LIN {X 0,Y 418.5,Z 298.346,A -85,B 0,C 180,E1 -10082.888,E2 -10082.888} C_VEL
LIN {X 0,Y 418.491,Z 298.347,A -85,B 0,C 180,E1 -10086.751,E2 -10086.751} C_VEL
LIN {X 0,Y 418.4,Z 298.365,A -85,B 0,C 180,E1 -10088.695,E2 -10088.695} C_VEL
LIN {X 0,Y 418.315,Z 298.368,A -85,B 0,C 180,E1 -10091.631,E2 -10091.631} C_VEL
LIN {X 0,Y 418.303,Z 298.378,A -85,B 0,C 180,E1 -10094.597,E2 -10094.597} C_VEL
LIN {X 0,Y 418.288,Z 298.376,A -85,B 0,C 180,E1 -10097.604,E2 -10097.604} C_VEL
LIN {X 0,Y 418.25,Z 298.383,A -85,B 0,C 180,E1 -10100.663,E2 -10100.663} C_VEL
LIN {X 0,Y 418.277,Z 298.377,A -85,B 0,C 180,E1 -10103.782,E2 -10103.782} C_VEL
LIN {X 0,Y 418.311,Z 298.378,A -85,B 0,C 180,E1 -10107.071,E2 -10107.071} C_VEL
LIN {X 0,Y 418.245,Z 298.383,A -85,B 0,C 180,E1 -10110.272,E2 -10110.272} C_VEL
LIN {X 0,Y 418.249,Z 298.384,A -85,B 0,C 180,E1 -10113.677,E2 -10113.677} C_VEL
LIN {X 0,Y 418.241,Z 298.389,A -85,B 0,C 180,E1 -10117.224,E2 -10117.224} C_VEL
LIN {X 0,Y 418.247,Z 298.372,A -85,B 0,C 180,E1 -10119.683,E2 -10119.683} C_VEL
LIN {X 0,Y 418.231,Z 298.384,A -85,B 0,C 180,E1 -10122.321,E2 -10122.321} C_VEL
LIN {X 0,Y 418.237,Z 298.386,A -85,B 0,C 180,E1 -10125.109,E2 -10125.109} C_VEL
LIN {X 0,Y 418.241,Z 298.389,A -85,B 0,C 180,E1 -10127.767,E2 -10127.767} C_VEL
LIN {X 0,Y 418.247,Z 298.383,A -85,B 0,C 180,E1 -10130.621,E2 -10130.621} C_VEL
LIN {X 0,Y 418.245,Z 298.389,A -85,B 0,C 180,E1 -10133.976,E2 -10133.976} C_VEL
LIN {X 0,Y 418.26,Z 298.385,A -85,B 0,C 180,E1 -10137.156,E2 -10137.156} C_VEL
LIN {X 0,Y 418.271,Z 298.384,A -85,B 0,C 180,E1 -10140.896,E2 -10140.896} C_VEL
LIN {X 0,Y 418.35,Z 298.445,A -85,B 0,C 180,E1 -10141.77,E2 -10141.77} C_VEL
LIN {X 0,Y 421.032,Z 311.046,A -85,B 0,C 180,E1 -10144.57,E2 -10144.57} C_VEL
LIN {X 0,Y 421.704,Z 316.103,A -85,B 0,C 180,E1 -10145.639,E2 -10145.639} C_VEL
LIN {X 0,Y 420.393,Z 334.263,A -85,B 0,C 180,E1 -10149.191,E2 -10149.191} C_VEL
LIN {X 0,Y 419.959,Z 341.409,A -85,B 0,C 180,E1 -10150.575,E2 -10150.575} C_VEL
LIN {X 0,Y 424.044,Z 365.211,A -85,B 0,C 180,E1 -10151.223,E2 -10151.223} C_VEL
LIN {X 0,Y 424.504,Z 369.379,A -85,B 0,C 180,E1 -10151.321,E2 -10151.321} C_VEL
LIN {X 0,Y 423.445,Z 450.649,A -85,B 0,C 180,E1 -10152.742,E2 -10152.742} C_VEL
LIN {X 0,Y 422.844,Z 463.629,A -85,B 0,C 180,E1 -10153.152,E2 -10153.152} C_VEL
LIN {X 0,Y 422.218,Z 476.184,A -85,B 0,C 180,E1 -10153.748,E2 -10153.748} C_VEL
LIN {X 0,Y 421.378,Z 488.172,A -85,B 0,C 180,E1 -10154.522,E2 -10154.522} C_VEL
LIN {X 0,Y 420.526,Z 499.632,A -85,B 0,C 180,E1 -10155.482,E2 -10155.482} C_VEL
LIN {X 0,Y 419.746,Z 509.977,A -85,B 0,C 180,E1 -10156.566,E2 -10156.566} C_VEL
LIN {X 0,Y 419.111,Z 518.454,A -85,B 0,C 180,E1 -10157.654,E2 -10157.654} C_VEL
LIN {X 0,Y 418.291,Z 527.665,A -85,B 0,C 180,E1 -10159.104,E2 -10159.104} C_VEL
LIN {X 0,Y 417.766,Z 535.087,A -85,B 0,C 180,E1 -10160.559,E2 -10160.559} C_VEL
LIN {X 0,Y 417.368,Z 541.95,A -85,B 0,C 180,E1 -10162.258,E2 -10162.258} C_VEL
LIN {X 0,Y 417.137,Z 546.573,A -85,B 0,C 180,E1 -10163.745,E2 -10163.745} C_VEL
LIN {X 0,Y 417.107,Z 549.952,A -85,B 0,C 180,E1 -10165.167,E2 -10165.167} C_VEL
LIN {X 0,Y 417.03,Z 553.007,A -85,B 0,C 180,E1 -10167.102,E2 -10167.102} C_VEL
LIN {X 0,Y 417.07,Z 553.941,A -85,B 0,C 180,E1 -10168.068,E2 -10168.068} C_VEL
LIN {X 0,Y 417.013,Z 554.471,A -85,B 0,C 180,E1 -10169.034,E2 -10169.034} C_VEL
LIN {X 0,Y 417.027,Z 554.572,A -85,B 0,C 180,E1 -10170,E2 -10170} C_VEL
LIN {X 0,Y 417.072,Z 553.609,A -85,B 0,C 180,E1 -10171.931,E2 -10171.931} C_VEL
LIN {X 0,Y 417.061,Z 552.532,A -85,B 0,C 180,E1 -10172.897,E2 -10172.897} C_VEL
LIN {X 0,Y 417.018,Z 550.996,A -85,B 0,C 180,E1 -10173.865,E2 -10173.865} C_VEL
LIN {X 0,Y 417.119,Z 547.906,A -85,B 0,C 180,E1 -10175.317,E2 -10175.317} C_VEL
LIN {X 0,Y 417.231,Z 543.743,A -85,B 0,C 180,E1 -10176.771,E2 -10176.771} C_VEL
LIN {X 0,Y 417.481,Z 537.373,A -85,B 0,C 180,E1 -10178.47,E2 -10178.47} C_VEL
LIN {X 0,Y 417.858,Z 530.43,A -85,B 0,C 180,E1 -10179.927,E2 -10179.927} C_VEL
LIN {X 0,Y 418.281,Z 523.332,A -85,B 0,C 180,E1 -10181.141,E2 -10181.141} C_VEL
LIN {X 0,Y 418.878,Z 514.765,A -85,B 0,C 180,E1 -10182.352,E2 -10182.352} C_VEL
LIN {X 0,Y 419.513,Z 504.16,A -85,B 0,C 180,E1 -10183.564,E2 -10183.564} C_VEL
LIN {X 0,Y 420.15,Z 493.654,A -85,B 0,C 180,E1 -10184.531,E2 -10184.531} C_VEL
LIN {X 0,Y 420.876,Z 482.102,A -85,B 0,C 180,E1 -10185.372,E2 -10185.372} C_VEL
LIN {X 0,Y 421.506,Z 470.115,A -85,B 0,C 180,E1 -10186.03,E2 -10186.03} C_VEL
LIN {X 0,Y 422.019,Z 457.151,A -85,B 0,C 180,E1 -10186.538,E2 -10186.538} C_VEL
LIN {X 0,Y 422.375,Z 445.077,A -85,B 0,C 180,E1 -10186.835,E2 -10186.835} C_VEL
LIN {X 0,Y 423.05,Z 367.123,A -85,B 0,C 180,E1 -10188.161,E2 -10188.161} C_VEL
LIN {X 0,Y 419.349,Z 341.69,A -85,B 0,C 180,E1 -10188.757,E2 -10188.757} C_VEL
LIN {X 0,Y 420.441,Z 322.825,A -85,B 0,C 180,E1 -10192.351,E2 -10192.351} C_VEL
LIN {X 0,Y 420.939,Z 312.172,A -85,B 0,C 180,E1 -10194.407,E2 -10194.407} C_VEL
LIN {X 0,Y 418.487,Z 299.135,A -85,B 0,C 180,E1 -10197.117,E2 -10197.117} C_VEL
LIN {X 0,Y 418.338,Z 298.378,A -85,B 0,C 180,E1 -10197.322,E2 -10197.322} C_VEL
LIN {X 0,Y 418.239,Z 298.384,A -85,B 0,C 180,E1 -10201.019,E2 -10201.019} C_VEL
LIN {X 0,Y 418.248,Z 298.383,A -85,B 0,C 180,E1 -10203.676,E2 -10203.676} C_VEL
LIN {X 0,Y 418.238,Z 298.383,A -85,B 0,C 180,E1 -10207.223,E2 -10207.223} C_VEL
LIN {X 0,Y 418.243,Z 298.383,A -85,B 0,C 180,E1 -10209.682,E2 -10209.682} C_VEL
LIN {X 0,Y 418.228,Z 298.391,A -85,B 0,C 180,E1 -10212.32,E2 -10212.32} C_VEL
LIN {X 0,Y 418.233,Z 298.384,A -85,B 0,C 180,E1 -10215.108,E2 -10215.108} C_VEL
LIN {X 0,Y 418.238,Z 298.383,A -85,B 0,C 180,E1 -10217.766,E2 -10217.766} C_VEL
LIN {X 0,Y 418.253,Z 298.389,A -85,B 0,C 180,E1 -10220.618,E2 -10220.618} C_VEL
LIN {X 0,Y 418.24,Z 298.383,A -85,B 0,C 180,E1 -10223.975,E2 -10223.975} C_VEL
LIN {X 0,Y 418.254,Z 298.384,A -85,B 0,C 180,E1 -10227.155,E2 -10227.155} C_VEL
LIN {X 0,Y 418.265,Z 298.387,A -85,B 0,C 180,E1 -10230.895,E2 -10230.895} C_VEL
LIN {X 0,Y 418.267,Z 298.379,A -85,B 0,C 180,E1 -10234.095,E2 -10234.095} C_VEL
LIN {X 0,Y 418.234,Z 298.389,A -85,B 0,C 180,E1 -10237.263,E2 -10237.263} C_VEL
LIN {X 0,Y 418.279,Z 298.378,A -85,B 0,C 180,E1 -10240.364,E2 -10240.364} C_VEL
LIN {X 0,Y 418.313,Z 298.38,A -85,B 0,C 180,E1 -10243.404,E2 -10243.404} C_VEL
LIN {X 0,Y 418.341,Z 298.373,A -85,B 0,C 180,E1 -10246.999,E2 -10246.999} C_VEL
LIN {X 0,Y 418.336,Z 298.37,A -85,B 0,C 180,E1 -10250.328,E2 -10250.328} C_VEL
LIN {X 0,Y 418.487,Z 298.356,A -85,B 0,C 180,E1 -10253.249,E2 -10253.249} C_VEL
LIN {X 0,Y 418.333,Z 298.374,A -85,B 0,C 180,E1 -10255.181,E2 -10255.181} C_VEL
LIN {X 0,Y 418.536,Z 298.348,A -85,B 0,C 180,E1 -10258.075,E2 -10258.075} C_VEL
LIN {X 0,Y 418.665,Z 298.334,A -85,B 0,C 180,E1 -10260,E2 -10260} C_VEL
LIN {X 0,Y 418.496,Z 298.35,A -85,B 0,C 180,E1 -10262.888,E2 -10262.888} C_VEL
LIN {X 0,Y 418.452,Z 298.356,A -85,B 0,C 180,E1 -10266.52,E2 -10266.52} C_VEL
LIN {X 0,Y 418.335,Z 298.374,A -85,B 0,C 180,E1 -10269.671,E2 -10269.671} C_VEL
LIN {X 0,Y 418.341,Z 298.37,A -85,B 0,C 180,E1 -10273.001,E2 -10273.001} C_VEL
LIN {X 0,Y 418.307,Z 298.376,A -85,B 0,C 180,E1 -10276.735,E2 -10276.735} C_VEL
LIN {X 0,Y 418.265,Z 298.382,A -85,B 0,C 180,E1 -10279.79,E2 -10279.79} C_VEL
LIN {X 0,Y 418.226,Z 298.387,A -85,B 0,C 180,E1 -10282.737,E2 -10282.737} C_VEL
LIN {X 0,Y 418.256,Z 298.382,A -85,B 0,C 180,E1 -10285.905,E2 -10285.905} C_VEL
LIN {X 0,Y 418.263,Z 298.381,A -85,B 0,C 180,E1 -10289.105,E2 -10289.105} C_VEL
LIN {X 0,Y 418.252,Z 298.386,A -85,B 0,C 180,E1 -10292.844,E2 -10292.844} C_VEL
LIN {X 0,Y 418.24,Z 298.385,A -85,B 0,C 180,E1 -10296.238,E2 -10296.238} C_VEL
LIN {X 0,Y 418.24,Z 298.382,A -85,B 0,C 180,E1 -10299.683,E2 -10299.683} C_VEL
LIN {X 0,Y 418.225,Z 298.386,A -85,B 0,C 180,E1 -10302.321,E2 -10302.321} C_VEL
LIN {X 0,Y 418.231,Z 298.389,A -85,B 0,C 180,E1 -10305.109,E2 -10305.109} C_VEL
LIN {X 0,Y 418.219,Z 298.386,A -85,B 0,C 180,E1 -10307.765,E2 -10307.765} C_VEL
LIN {X 0,Y 418.236,Z 298.386,A -85,B 0,C 180,E1 -10311.557,E2 -10311.557} C_VEL
LIN {X 0,Y 418.254,Z 298.388,A -85,B 0,C 180,E1 -10315.159,E2 -10315.159} C_VEL
LIN {X 0,Y 418.242,Z 298.388,A -85,B 0,C 180,E1 -10317.472,E2 -10317.472} C_VEL
LIN {X 0,Y 418.258,Z 298.382,A -85,B 0,C 180,E1 -10320.898,E2 -10320.898} C_VEL
LIN {X 0,Y 418.221,Z 298.386,A -85,B 0,C 180,E1 -10324.093,E2 -10324.093} C_VEL
LIN {X 0,Y 418.225,Z 298.388,A -85,B 0,C 180,E1 -10327.264,E2 -10327.264} C_VEL
LIN {X 0,Y 418.281,Z 298.378,A -85,B 0,C 180,E1 -10330.365,E2 -10330.365} C_VEL
LIN {X 0,Y 418.314,Z 298.377,A -85,B 0,C 180,E1 -10333.405,E2 -10333.405} C_VEL
LIN {X 0,Y 418.344,Z 298.373,A -85,B 0,C 180,E1 -10337,E2 -10337} C_VEL
LIN {X 0,Y 418.402,Z 298.509,A -85,B 0,C 180,E1 -10338.218,E2 -10338.218} C_VEL
LIN {X 0,Y 419.848,Z 307.982,A -85,B 0,C 180,E1 -10340.364,E2 -10340.364} C_VEL
LIN {X 0,Y 419.769,Z 312.482,A -85,B 0,C 180,E1 -10341.334,E2 -10341.334} C_VEL
LIN {X 0,Y 423.405,Z 332.436,A -85,B 0,C 180,E1 -10341.834,E2 -10341.834} C_VEL
LIN {X 0,Y 422.377,Z 420.161,A -85,B 0,C 180,E1 -10343.342,E2 -10343.342} C_VEL
LIN {X 0,Y 422.005,Z 433.941,A -85,B 0,C 180,E1 -10343.786,E2 -10343.786} C_VEL
LIN {X 0,Y 421.617,Z 446.275,A -85,B 0,C 180,E1 -10344.38,E2 -10344.38} C_VEL
LIN {X 0,Y 421.232,Z 455.15,A -85,B 0,C 180,E1 -10344.942,E2 -10344.942} C_VEL
LIN {X 0,Y 420.359,Z 458.68,A -85,B 0,C 180,E1 -10345.169,E2 -10345.169} C_VEL
LIN {X 0,Y 417.152,Z 464.137,A -85,B 0,C 180,E1 -10345.503,E2 -10345.503} C_VEL
LIN {X 0,Y 413.955,Z 469.396,A -85,B 0,C 180,E1 -10345.888,E2 -10345.888} C_VEL
LIN {X 0,Y 413.101,Z 472.61,A -85,B 0,C 180,E1 -10346.19,E2 -10346.19} C_VEL
LIN {X 0,Y 412.334,Z 482.525,A -85,B 0,C 180,E1 -10347.314,E2 -10347.314} C_VEL
LIN {X 0,Y 411.859,Z 491.264,A -85,B 0,C 180,E1 -10348.534,E2 -10348.534} C_VEL
LIN {X 0,Y 411.253,Z 499.825,A -85,B 0,C 180,E1 -10350,E2 -10350} C_VEL
LIN {X 0,Y 410.769,Z 506.671,A -85,B 0,C 180,E1 -10351.471,E2 -10351.471} C_VEL
LIN {X 0,Y 410.451,Z 512.158,A -85,B 0,C 180,E1 -10352.945,E2 -10352.945} C_VEL
LIN {X 0,Y 410.172,Z 516.476,A -85,B 0,C 180,E1 -10354.422,E2 -10354.422} C_VEL
LIN {X 0,Y 410.15,Z 519.723,A -85,B 0,C 180,E1 -10355.901,E2 -10355.901} C_VEL
LIN {X 0,Y 410.05,Z 521.347,A -85,B 0,C 180,E1 -10356.891,E2 -10356.891} C_VEL
LIN {X 0,Y 409.941,Z 522.573,A -85,B 0,C 180,E1 -10357.883,E2 -10357.883} C_VEL
LIN {X 0,Y 409.863,Z 523.362,A -85,B 0,C 180,E1 -10358.878,E2 -10358.878} C_VEL
LIN {X 0,Y 409.93,Z 523.73,A -85,B 0,C 180,E1 -10360.871,E2 -10360.871} C_VEL
LIN {X 0,Y 409.993,Z 523.009,A -85,B 0,C 180,E1 -10362.291,E2 -10362.291} C_VEL
LIN {X 0,Y 410.048,Z 521.225,A -85,B 0,C 180,E1 -10363.884,E2 -10363.884} C_VEL
LIN {X 0,Y 410.293,Z 518.521,A -85,B 0,C 180,E1 -10365.397,E2 -10365.397} C_VEL
LIN {X 0,Y 410.547,Z 514.751,A -85,B 0,C 180,E1 -10366.919,E2 -10366.919} C_VEL
LIN {X 0,Y 410.942,Z 509.796,A -85,B 0,C 180,E1 -10368.445,E2 -10368.445} C_VEL
LIN {X 0,Y 411.611,Z 502.906,A -85,B 0,C 180,E1 -10370.101,E2 -10370.101} C_VEL
LIN {X 0,Y 412.178,Z 495.548,A -85,B 0,C 180,E1 -10371.506,E2 -10371.506} C_VEL
LIN {X 0,Y 412.961,Z 487.353,A -85,B 0,C 180,E1 -10372.779,E2 -10372.779} C_VEL
LIN {X 0,Y 413.852,Z 477.278,A -85,B 0,C 180,E1 -10374.052,E2 -10374.052} C_VEL
LIN {X 0,Y 414.666,Z 467.31,A -85,B 0,C 180,E1 -10375.069,E2 -10375.069} C_VEL
LIN {X 0,Y 415.429,Z 456.392,A -85,B 0,C 180,E1 -10375.96,E2 -10375.96} C_VEL
LIN {X 0,Y 416.125,Z 444.455,A -85,B 0,C 180,E1 -10376.713,E2 -10376.713} C_VEL
LIN {X 0,Y 416.599,Z 431.865,A -85,B 0,C 180,E1 -10377.3,E2 -10377.3} C_VEL
LIN {X 0,Y 416.859,Z 420.649,A -85,B 0,C 180,E1 -10377.656,E2 -10377.656} C_VEL
LIN {X 0,Y 418.259,Z 333.539,A -85,B 0,C 180,E1 -10379.19,E2 -10379.19} C_VEL
LIN {X 0,Y 413.571,Z 313.012,A -85,B 0,C 180,E1 -10379.833,E2 -10379.833} C_VEL
LIN {X 0,Y 413.27,Z 309.221,A -85,B 0,C 180,E1 -10380.676,E2 -10380.676} C_VEL
LIN {X 0,Y 411.221,Z 299.263,A -85,B 0,C 180,E1 -10383.068,E2 -10383.068} C_VEL
LIN {X 0,Y 411.192,Z 299.263,A -85,B 0,C 180,E1 -10386.553,E2 -10386.553} C_VEL
LIN {X 0,Y 411.21,Z 299.263,A -85,B 0,C 180,E1 -10389.728,E2 -10389.728} C_VEL
LIN {X 0,Y 411.172,Z 299.267,A -85,B 0,C 180,E1 -10393.134,E2 -10393.134} C_VEL
LIN {X 0,Y 411.167,Z 299.266,A -85,B 0,C 180,E1 -10395.881,E2 -10395.881} C_VEL
LIN {X 0,Y 411.163,Z 299.27,A -85,B 0,C 180,E1 -10398.772,E2 -10398.772} C_VEL
LIN {X 0,Y 411.205,Z 299.257,A -85,B 0,C 180,E1 -10401.831,E2 -10401.831} C_VEL
LIN {X 0,Y 411.21,Z 299.261,A -85,B 0,C 180,E1 -10405.122,E2 -10405.122} C_VEL
LIN {X 0,Y 411.165,Z 299.26,A -85,B 0,C 180,E1 -10408.003,E2 -10408.003} C_VEL
LIN {X 0,Y 411.217,Z 299.256,A -85,B 0,C 180,E1 -10411.41,E2 -10411.41} C_VEL
LIN {X 0,Y 411.236,Z 299.255,A -85,B 0,C 180,E1 -10413.619,E2 -10413.619} C_VEL
LIN {X 0,Y 411.196,Z 299.256,A -85,B 0,C 180,E1 -10416.852,E2 -10416.852} C_VEL
LIN {X 0,Y 411.214,Z 299.253,A -85,B 0,C 180,E1 -10420.051,E2 -10420.051} C_VEL
LIN {X 0,Y 411.262,Z 299.256,A -85,B 0,C 180,E1 -10423.131,E2 -10423.131} C_VEL
LIN {X 0,Y 411.305,Z 299.248,A -85,B 0,C 180,E1 -10426.896,E2 -10426.896} C_VEL
LIN {X 0,Y 411.292,Z 299.251,A -85,B 0,C 180,E1 -10430.161,E2 -10430.161} C_VEL
LIN {X 0,Y 411.482,Z 299.226,A -85,B 0,C 180,E1 -10432.147,E2 -10432.147} C_VEL
LIN {X 0,Y 411.471,Z 299.229,A -85,B 0,C 180,E1 -10434.118,E2 -10434.118} C_VEL
LIN {X 0,Y 411.511,Z 299.221,A -85,B 0,C 180,E1 -10438.043,E2 -10438.043} C_VEL
LIN {X 0,Y 411.64,Z 299.21,A -85,B 0,C 180,E1 -10440,E2 -10440} C_VEL
LIN {X 0,Y 411.457,Z 299.223,A -85,B 0,C 180,E1 -10442.937,E2 -10442.937} C_VEL
LIN {X 0,Y 411.458,Z 299.222,A -85,B 0,C 180,E1 -10446.867,E2 -10446.867} C_VEL
LIN {X 0,Y 411.354,Z 299.241,A -85,B 0,C 180,E1 -10448.845,E2 -10448.845} C_VEL
LIN {X 0,Y 411.283,Z 299.245,A -85,B 0,C 180,E1 -10451.833,E2 -10451.833} C_VEL
LIN {X 0,Y 411.26,Z 299.252,A -85,B 0,C 180,E1 -10454.853,E2 -10454.853} C_VEL
LIN {X 0,Y 411.253,Z 299.253,A -85,B 0,C 180,E1 -10457.915,E2 -10457.915} C_VEL
LIN {X 0,Y 411.197,Z 299.263,A -85,B 0,C 180,E1 -10461.034,E2 -10461.034} C_VEL
LIN {X 0,Y 411.221,Z 299.257,A -85,B 0,C 180,E1 -10464.216,E2 -10464.216} C_VEL
LIN {X 0,Y 411.26,Z 299.253,A -85,B 0,C 180,E1 -10467.478,E2 -10467.478} C_VEL
LIN {X 0,Y 411.19,Z 299.268,A -85,B 0,C 180,E1 -10470.848,E2 -10470.848} C_VEL
LIN {X 0,Y 411.206,Z 299.26,A -85,B 0,C 180,E1 -10474.334,E2 -10474.334} C_VEL
LIN {X 0,Y 411.194,Z 299.261,A -85,B 0,C 180,E1 -10477.974,E2 -10477.974} C_VEL
LIN {X 0,Y 411.165,Z 299.255,A -85,B 0,C 180,E1 -10481.229,E2 -10481.229} C_VEL
LIN {X 0,Y 411.177,Z 299.262,A -85,B 0,C 180,E1 -10484.491,E2 -10484.491} C_VEL
LIN {X 0,Y 411.178,Z 299.265,A -85,B 0,C 180,E1 -10488.195,E2 -10488.195} C_VEL
LIN {X 0,Y 411.212,Z 299.259,A -85,B 0,C 180,E1 -10490.775,E2 -10490.775} C_VEL
LIN {X 0,Y 411.2,Z 299.263,A -85,B 0,C 180,E1 -10494.471,E2 -10494.471} C_VEL
LIN {X 0,Y 411.21,Z 299.263,A -85,B 0,C 180,E1 -10496.873,E2 -10496.873} C_VEL
LIN {X 0,Y 411.235,Z 299.26,A -85,B 0,C 180,E1 -10500.644,E2 -10500.644} C_VEL
LIN {X 0,Y 411.293,Z 299.263,A -85,B 0,C 180,E1 -10501.416,E2 -10501.416} C_VEL
LIN {X 0,Y 413.882,Z 311.315,A -85,B 0,C 180,E1 -10504.156,E2 -10504.156} C_VEL
LIN {X 0,Y 414.812,Z 317.388,A -85,B 0,C 180,E1 -10505.475,E2 -10505.475} C_VEL
LIN {X 0,Y 413.452,Z 335.534,A -85,B 0,C 180,E1 -10509.086,E2 -10509.086} C_VEL
LIN {X 0,Y 413.097,Z 341.103,A -85,B 0,C 180,E1 -10510.184,E2 -10510.184} C_VEL
LIN {X 0,Y 417.21,Z 364.546,A -85,B 0,C 180,E1 -10510.848,E2 -10510.848} C_VEL
LIN {X 0,Y 417.876,Z 371.311,A -85,B 0,C 180,E1 -10511.007,E2 -10511.007} C_VEL
LIN {X 0,Y 416.813,Z 449.726,A -85,B 0,C 180,E1 -10512.395,E2 -10512.395} C_VEL
LIN {X 0,Y 416.15,Z 462.924,A -85,B 0,C 180,E1 -10512.81,E2 -10512.81} C_VEL
LIN {X 0,Y 415.502,Z 475.585,A -85,B 0,C 180,E1 -10513.415,E2 -10513.415} C_VEL
LIN {X 0,Y 414.683,Z 486.873,A -85,B 0,C 180,E1 -10514.14,E2 -10514.14} C_VEL
LIN {X 0,Y 413.765,Z 498.523,A -85,B 0,C 180,E1 -10515.113,E2 -10515.113} C_VEL
LIN {X 0,Y 412.88,Z 509.01,A -85,B 0,C 180,E1 -10516.213,E2 -10516.213} C_VEL
LIN {X 0,Y 412.154,Z 518.486,A -85,B 0,C 180,E1 -10517.443,E2 -10517.443} C_VEL
LIN {X 0,Y 411.307,Z 527.627,A -85,B 0,C 180,E1 -10518.917,E2 -10518.917} C_VEL
LIN {X 0,Y 410.741,Z 535.006,A -85,B 0,C 180,E1 -10520.396,E2 -10520.396} C_VEL
LIN {X 0,Y 410.322,Z 541.816,A -85,B 0,C 180,E1 -10522.124,E2 -10522.124} C_VEL
LIN {X 0,Y 410.043,Z 546.76,A -85,B 0,C 180,E1 -10523.776,E2 -10523.776} C_VEL
LIN {X 0,Y 410.019,Z 549.761,A -85,B 0,C 180,E1 -10525.083,E2 -10525.083} C_VEL
LIN {X 0,Y 409.928,Z 552.786,A -85,B 0,C 180,E1 -10527.051,E2 -10527.051} C_VEL
LIN {X 0,Y 409.997,Z 553.709,A -85,B 0,C 180,E1 -10528.035,E2 -10528.035} C_VEL
LIN {X 0,Y 409.938,Z 554.216,A -85,B 0,C 180,E1 -10529.017,E2 -10529.017} C_VEL
LIN {X 0,Y 409.948,Z 554.301,A -85,B 0,C 180,E1 -10530,E2 -10530} C_VEL
LIN {X 0,Y 410.001,Z 553.314,A -85,B 0,C 180,E1 -10531.964,E2 -10531.964} C_VEL
LIN {X 0,Y 409.959,Z 552.213,A -85,B 0,C 180,E1 -10532.948,E2 -10532.948} C_VEL
LIN {X 0,Y 409.937,Z 550.661,A -85,B 0,C 180,E1 -10533.932,E2 -10533.932} C_VEL
LIN {X 0,Y 410.014,Z 547.54,A -85,B 0,C 180,E1 -10535.409,E2 -10535.409} C_VEL
LIN {X 0,Y 410.163,Z 543.347,A -85,B 0,C 180,E1 -10536.888,E2 -10536.888} C_VEL
LIN {X 0,Y 410.413,Z 536.942,A -85,B 0,C 180,E1 -10538.617,E2 -10538.617} C_VEL
LIN {X 0,Y 410.8,Z 529.958,A -85,B 0,C 180,E1 -10540.099,E2 -10540.099} C_VEL
LIN {X 0,Y 411.381,Z 521.191,A -85,B 0,C 180,E1 -10541.58,E2 -10541.58} C_VEL
LIN {X 0,Y 411.996,Z 512.2,A -85,B 0,C 180,E1 -10542.812,E2 -10542.812} C_VEL
LIN {X 0,Y 412.588,Z 503.016,A -85,B 0,C 180,E1 -10543.847,E2 -10543.847} C_VEL
LIN {X 0,Y 413.22,Z 492.899,A -85,B 0,C 180,E1 -10544.78,E2 -10544.78} C_VEL
LIN {X 0,Y 414,Z 481.167,A -85,B 0,C 180,E1 -10545.634,E2 -10545.634} C_VEL
LIN {X 0,Y 414.609,Z 468.943,A -85,B 0,C 180,E1 -10546.304,E2 -10546.304} C_VEL
LIN {X 0,Y 415.215,Z 455.622,A -85,B 0,C 180,E1 -10546.817,E2 -10546.817} C_VEL
LIN {X 0,Y 415.558,Z 442.471,A -85,B 0,C 180,E1 -10547.12,E2 -10547.12} C_VEL
LIN {X 0,Y 416.225,Z 367.94,A -85,B 0,C 180,E1 -10548.406,E2 -10548.406} C_VEL
LIN {X 0,Y 412.405,Z 341.35,A -85,B 0,C 180,E1 -10549.053,E2 -10549.053} C_VEL
LIN {X 0,Y 413.456,Z 323.637,A -85,B 0,C 180,E1 -10552.485,E2 -10552.485} C_VEL
LIN {X 0,Y 414.045,Z 314.324,A -85,B 0,C 180,E1 -10554.306,E2 -10554.306} C_VEL
LIN {X 0,Y 412.136,Z 303.43,A -85,B 0,C 180,E1 -10556.591,E2 -10556.591} C_VEL
LIN {X 0,Y 411.314,Z 299.253,A -85,B 0,C 180,E1 -10557.507,E2 -10557.507} C_VEL
LIN {X 0,Y 411.189,Z 299.264,A -85,B 0,C 180,E1 -10560.847,E2 -10560.847} C_VEL
LIN {X 0,Y 411.206,Z 299.265,A -85,B 0,C 180,E1 -10564.333,E2 -10564.333} C_VEL
LIN {X 0,Y 411.19,Z 299.264,A -85,B 0,C 180,E1 -10567.973,E2 -10567.973} C_VEL
LIN {X 0,Y 411.162,Z 299.264,A -85,B 0,C 180,E1 -10571.228,E2 -10571.228} C_VEL
LIN {X 0,Y 411.174,Z 299.271,A -85,B 0,C 180,E1 -10574.49,E2 -10574.49} C_VEL
LIN {X 0,Y 411.175,Z 299.266,A -85,B 0,C 180,E1 -10578.194,E2 -10578.194} C_VEL
LIN {X 0,Y 411.217,Z 299.264,A -85,B 0,C 180,E1 -10580.775,E2 -10580.775} C_VEL
LIN {X 0,Y 411.195,Z 299.264,A -85,B 0,C 180,E1 -10584.471,E2 -10584.471} C_VEL
LIN {X 0,Y 411.204,Z 299.266,A -85,B 0,C 180,E1 -10586.873,E2 -10586.873} C_VEL
LIN {X 0,Y 411.229,Z 299.26,A -85,B 0,C 180,E1 -10590.644,E2 -10590.644} C_VEL
LIN {X 0,Y 411.234,Z 299.256,A -85,B 0,C 180,E1 -10593.619,E2 -10593.619} C_VEL
LIN {X 0,Y 411.199,Z 299.264,A -85,B 0,C 180,E1 -10596.852,E2 -10596.852} C_VEL
LIN {X 0,Y 411.21,Z 299.258,A -85,B 0,C 180,E1 -10600.05,E2 -10600.05} C_VEL
LIN {X 0,Y 411.259,Z 299.258,A -85,B 0,C 180,E1 -10603.131,E2 -10603.131} C_VEL
LIN {X 0,Y 411.301,Z 299.249,A -85,B 0,C 180,E1 -10606.895,E2 -10606.895} C_VEL
LIN {X 0,Y 411.288,Z 299.249,A -85,B 0,C 180,E1 -10610.161,E2 -10610.161} C_VEL
LIN {X 0,Y 411.45,Z 299.231,A -85,B 0,C 180,E1 -10613.133,E2 -10613.133} C_VEL
LIN {X 0,Y 411.304,Z 299.249,A -85,B 0,C 180,E1 -10615.099,E2 -10615.099} C_VEL
LIN {X 0,Y 411.505,Z 299.225,A -85,B 0,C 180,E1 -10618.042,E2 -10618.042} C_VEL
LIN {X 0,Y 411.634,Z 299.21,A -85,B 0,C 180,E1 -10620,E2 -10620} C_VEL
LIN {X 0,Y 411.453,Z 299.228,A -85,B 0,C 180,E1 -10622.937,E2 -10622.937} C_VEL
LIN {X 0,Y 411.417,Z 299.234,A -85,B 0,C 180,E1 -10626.517,E2 -10626.517} C_VEL
LIN {X 0,Y 411.287,Z 299.254,A -85,B 0,C 180,E1 -10629.839,E2 -10629.839} C_VEL
LIN {X 0,Y 411.3,Z 299.247,A -85,B 0,C 180,E1 -10633.104,E2 -10633.104} C_VEL
LIN {X 0,Y 411.252,Z 299.254,A -85,B 0,C 180,E1 -10636.889,E2 -10636.889} C_VEL
LIN {X 0,Y 411.225,Z 299.26,A -85,B 0,C 180,E1 -10639.987,E2 -10639.987} C_VEL
LIN {X 0,Y 411.19,Z 299.261,A -85,B 0,C 180,E1 -10643.148,E2 -10643.148} C_VEL
LIN {X 0,Y 411.228,Z 299.263,A -85,B 0,C 180,E1 -10646.381,E2 -10646.381} C_VEL
LIN {X 0,Y 411.195,Z 299.26,A -85,B 0,C 180,E1 -10649.713,E2 -10649.713} C_VEL
LIN {X 0,Y 411.201,Z 299.261,A -85,B 0,C 180,E1 -10653.156,E2 -10653.156} C_VEL
LIN {X 0,Y 411.187,Z 299.267,A -85,B 0,C 180,E1 -10656.553,E2 -10656.553} C_VEL
LIN {X 0,Y 411.204,Z 299.259,A -85,B 0,C 180,E1 -10659.727,E2 -10659.727} C_VEL
LIN {X 0,Y 411.168,Z 299.268,A -85,B 0,C 180,E1 -10663.134,E2 -10663.134} C_VEL
LIN {X 0,Y 411.16,Z 299.264,A -85,B 0,C 180,E1 -10665.882,E2 -10665.882} C_VEL
LIN {X 0,Y 411.146,Z 299.27,A -85,B 0,C 180,E1 -10668.774,E2 -10668.774} C_VEL
LIN {X 0,Y 411.184,Z 299.262,A -85,B 0,C 180,E1 -10672.026,E2 -10672.026} C_VEL
LIN {X 0,Y 411.201,Z 299.262,A -85,B 0,C 180,E1 -10675.667,E2 -10675.667} C_VEL
LIN {X 0,Y 411.186,Z 299.267,A -85,B 0,C 180,E1 -10679.153,E2 -10679.153} C_VEL
LIN {X 0,Y 411.174,Z 299.271,A -85,B 0,C 180,E1 -10681.407,E2 -10681.407} C_VEL
LIN {X 0,Y 411.185,Z 299.263,A -85,B 0,C 180,E1 -10684.942,E2 -10684.942} C_VEL
LIN {X 0,Y 411.201,Z 299.263,A -85,B 0,C 180,E1 -10687.914,E2 -10687.914} C_VEL
LIN {X 0,Y 411.216,Z 299.259,A -85,B 0,C 180,E1 -10691.052,E2 -10691.052} C_VEL
LIN {X 0,Y 411.252,Z 299.258,A -85,B 0,C 180,E1 -10694.132,E2 -10694.132} C_VEL
LIN {X 0,Y 411.349,Z 299.328,A -85,B 0,C 180,E1 -10698.013,E2 -10698.013} C_VEL
LIN {X 0,Y 412.876,Z 308.819,A -85,B 0,C 180,E1 -10700.2,E2 -10700.2} C_VEL
LIN {X 0,Y 412.847,Z 313.009,A -85,B 0,C 180,E1 -10701.069,E2 -10701.069} C_VEL
LIN {X 0,Y 416.598,Z 333.572,A -85,B 0,C 180,E1 -10701.586,E2 -10701.586} C_VEL
LIN {X 0,Y 415.512,Z 420.703,A -85,B 0,C 180,E1 -10703.109,E2 -10703.109} C_VEL
LIN {X 0,Y 415.124,Z 434.395,A -85,B 0,C 180,E1 -10703.561,E2 -10703.561} C_VEL
LIN {X 0,Y 414.715,Z 446.675,A -85,B 0,C 180,E1 -10704.165,E2 -10704.165} C_VEL
LIN {X 0,Y 414.16,Z 457.694,A -85,B 0,C 180,E1 -10704.889,E2 -10704.889} C_VEL
LIN {X 0,Y 413.359,Z 467.932,A -85,B 0,C 180,E1 -10705.735,E2 -10705.735} C_VEL
LIN {X 0,Y 413.101,Z 472.61,A -85,B 0,C 180,E1 -10706.19,E2 -10706.19} C_VEL
LIN {X 0,Y 412.195,Z 477.351,A -85,B 0,C 180,E1 -10706.68,E2 -10706.68} C_VEL
LIN {X 0,Y 408.853,Z 484.704,A -85,B 0,C 180,E1 -10707.491,E2 -10707.491} C_VEL
LIN {X 0,Y 405.502,Z 491.482,A -85,B 0,C 180,E1 -10708.387,E2 -10708.387} C_VEL
LIN {X 0,Y 404.583,Z 495.318,A -85,B 0,C 180,E1 -10708.998,E2 -10708.998} C_VEL
LIN {X 0,Y 403.946,Z 503.177,A -85,B 0,C 180,E1 -10710.499,E2 -10710.499} C_VEL
LIN {X 0,Y 403.538,Z 509.415,A -85,B 0,C 180,E1 -10711.996,E2 -10711.996} C_VEL
LIN {X 0,Y 403.28,Z 514.384,A -85,B 0,C 180,E1 -10713.497,E2 -10713.497} C_VEL
LIN {X 0,Y 403.106,Z 518.239,A -85,B 0,C 180,E1 -10715.001,E2 -10715.001} C_VEL
LIN {X 0,Y 403.074,Z 520.846,A -85,B 0,C 180,E1 -10716.358,E2 -10716.358} C_VEL
LIN {X 0,Y 402.836,Z 522.968,A -85,B 0,C 180,E1 -10718.023,E2 -10718.023} C_VEL
LIN {X 0,Y 402.753,Z 524.028,A -85,B 0,C 180,E1 -10720.05,E2 -10720.05} C_VEL
LIN {X 0,Y 402.837,Z 523.975,A -85,B 0,C 180,E1 -10721.064,E2 -10721.064} C_VEL
LIN {X 0,Y 402.925,Z 523.275,A -85,B 0,C 180,E1 -10722.373,E2 -10722.373} C_VEL
LIN {X 0,Y 402.986,Z 521.296,A -85,B 0,C 180,E1 -10724.132,E2 -10724.132} C_VEL
LIN {X 0,Y 403.263,Z 518.501,A -85,B 0,C 180,E1 -10725.672,E2 -10725.672} C_VEL
LIN {X 0,Y 403.559,Z 514.633,A -85,B 0,C 180,E1 -10727.221,E2 -10727.221} C_VEL
LIN {X 0,Y 404.018,Z 509.574,A -85,B 0,C 180,E1 -10728.773,E2 -10728.773} C_VEL
LIN {X 0,Y 404.659,Z 503.152,A -85,B 0,C 180,E1 -10730.326,E2 -10730.326} C_VEL
LIN {X 0,Y 405.352,Z 495.012,A -85,B 0,C 180,E1 -10731.887,E2 -10731.887} C_VEL
LIN {X 0,Y 406.195,Z 486.657,A -85,B 0,C 180,E1 -10733.18,E2 -10733.18} C_VEL
LIN {X 0,Y 407.152,Z 476.377,A -85,B 0,C 180,E1 -10734.474,E2 -10734.474} C_VEL
LIN {X 0,Y 407.997,Z 466.069,A -85,B 0,C 180,E1 -10735.508,E2 -10735.508} C_VEL
LIN {X 0,Y 408.836,Z 454.76,A -85,B 0,C 180,E1 -10736.411,E2 -10736.411} C_VEL
LIN {X 0,Y 409.549,Z 442.103,A -85,B 0,C 180,E1 -10737.187,E2 -10737.187} C_VEL
LIN {X 0,Y 410.004,Z 429.317,A -85,B 0,C 180,E1 -10737.742,E2 -10737.742} C_VEL
LIN {X 0,Y 410.324,Z 419.457,A -85,B 0,C 180,E1 -10738.031,E2 -10738.031} C_VEL
LIN {X 0,Y 411.721,Z 334.697,A -85,B 0,C 180,E1 -10739.538,E2 -10739.538} C_VEL
LIN {X 0,Y 407.005,Z 314.386,A -85,B 0,C 180,E1 -10740.197,E2 -10740.197} C_VEL
LIN {X 0,Y 406.707,Z 313.102,A -85,B 0,C 180,E1 -10740.254,E2 -10740.254} C_VEL
LIN {X 0,Y 405.303,Z 305.327,A -85,B 0,C 180,E1 -10742.124,E2 -10742.124} C_VEL
LIN {X 0,Y 404.168,Z 300.142,A -85,B 0,C 180,E1 -10743.419,E2 -10743.419} C_VEL
LIN {X 0,Y 404.141,Z 300.146,A -85,B 0,C 180,E1 -10746.246,E2 -10746.246} C_VEL
LIN {X 0,Y 404.152,Z 300.145,A -85,B 0,C 180,E1 -10748.757,E2 -10748.757} C_VEL
LIN {X 0,Y 404.122,Z 300.144,A -85,B 0,C 180,E1 -10751.6,E2 -10751.6} C_VEL
LIN {X 0,Y 404.144,Z 300.142,A -85,B 0,C 180,E1 -10754.522,E2 -10754.522} C_VEL
LIN {X 0,Y 404.136,Z 300.142,A -85,B 0,C 180,E1 -10757.296,E2 -10757.296} C_VEL
LIN {X 0,Y 404.168,Z 300.136,A -85,B 0,C 180,E1 -10759.955,E2 -10759.955} C_VEL
LIN {X 0,Y 404.136,Z 300.142,A -85,B 0,C 180,E1 -10763.125,E2 -10763.125} C_VEL
LIN {X 0,Y 404.144,Z 300.136,A -85,B 0,C 180,E1 -10766.188,E2 -10766.188} C_VEL
LIN {X 0,Y 404.145,Z 300.135,A -85,B 0,C 180,E1 -10769.715,E2 -10769.715} C_VEL
LIN {X 0,Y 404.194,Z 300.13,A -85,B 0,C 180,E1 -10773.123,E2 -10773.123} C_VEL
LIN {X 0,Y 404.173,Z 300.135,A -85,B 0,C 180,E1 -10775.334,E2 -10775.334} C_VEL
LIN {X 0,Y 404.137,Z 300.139,A -85,B 0,C 180,E1 -10778.581,E2 -10778.581} C_VEL
LIN {X 0,Y 404.209,Z 300.135,A -85,B 0,C 180,E1 -10781.762,E2 -10781.762} C_VEL
LIN {X 0,Y 404.205,Z 300.128,A -85,B 0,C 180,E1 -10784.882,E2 -10784.882} C_VEL
LIN {X 0,Y 404.255,Z 300.126,A -85,B 0,C 180,E1 -10787.959,E2 -10787.959} C_VEL
LIN {X 0,Y 404.433,Z 300.104,A -85,B 0,C 180,E1 -10792.1,E2 -10792.1} C_VEL
LIN {X 0,Y 404.42,Z 300.106,A -85,B 0,C 180,E1 -10794.015,E2 -10794.015} C_VEL
LIN {X 0,Y 404.48,Z 300.096,A -85,B 0,C 180,E1 -10798.009,E2 -10798.009} C_VEL
LIN {X 0,Y 404.609,Z 300.086,A -85,B 0,C 180,E1 -10800,E2 -10800} C_VEL
LIN {X 0,Y 404.415,Z 300.1,A -85,B 0,C 180,E1 -10802.989,E2 -10802.989} C_VEL
LIN {X 0,Y 404.41,Z 300.099,A -85,B 0,C 180,E1 -10806.988,E2 -10806.988} C_VEL
LIN {X 0,Y 404.258,Z 300.127,A -85,B 0,C 180,E1 -10810.012,E2 -10810.012} C_VEL
LIN {X 0,Y 404.267,Z 300.123,A -85,B 0,C 180,E1 -10813.212,E2 -10813.212} C_VEL
LIN {X 0,Y 404.216,Z 300.131,A -85,B 0,C 180,E1 -10817.007,E2 -10817.007} C_VEL
LIN {X 0,Y 404.164,Z 300.136,A -85,B 0,C 180,E1 -10820.352,E2 -10820.352} C_VEL
LIN {X 0,Y 404.164,Z 300.135,A -85,B 0,C 180,E1 -10823.575,E2 -10823.575} C_VEL
LIN {X 0,Y 404.184,Z 300.134,A -85,B 0,C 180,E1 -10825.767,E2 -10825.767} C_VEL
LIN {X 0,Y 404.196,Z 300.131,A -85,B 0,C 180,E1 -10828,E2 -10828} C_VEL
LIN {X 0,Y 404.14,Z 300.139,A -85,B 0,C 180,E1 -10831.558,E2 -10831.558} C_VEL
LIN {X 0,Y 404.185,Z 300.138,A -85,B 0,C 180,E1 -10835.016,E2 -10835.016} C_VEL
LIN {X 0,Y 404.153,Z 300.14,A -85,B 0,C 180,E1 -10838.757,E2 -10838.757} C_VEL
LIN {X 0,Y 404.124,Z 300.137,A -85,B 0,C 180,E1 -10841.6,E2 -10841.6} C_VEL
LIN {X 0,Y 404.147,Z 300.138,A -85,B 0,C 180,E1 -10844.522,E2 -10844.522} C_VEL
LIN {X 0,Y 404.138,Z 300.144,A -85,B 0,C 180,E1 -10847.296,E2 -10847.296} C_VEL
LIN {X 0,Y 404.171,Z 300.139,A -85,B 0,C 180,E1 -10849.956,E2 -10849.956} C_VEL
LIN {X 0,Y 404.138,Z 300.138,A -85,B 0,C 180,E1 -10853.125,E2 -10853.125} C_VEL
LIN {X 0,Y 404.147,Z 300.145,A -85,B 0,C 180,E1 -10856.188,E2 -10856.188} C_VEL
LIN {X 0,Y 404.148,Z 300.142,A -85,B 0,C 180,E1 -10859.715,E2 -10859.715} C_VEL
LIN {X 0,Y 404.228,Z 300.25,A -85,B 0,C 180,E1 -10861.082,E2 -10861.082} C_VEL
LIN {X 0,Y 406.936,Z 312.373,A -85,B 0,C 180,E1 -10863.906,E2 -10863.906} C_VEL
LIN {X 0,Y 407.939,Z 318.68,A -85,B 0,C 180,E1 -10865.305,E2 -10865.305} C_VEL
LIN {X 0,Y 406.646,Z 335.519,A -85,B 0,C 180,E1 -10868.719,E2 -10868.719} C_VEL
LIN {X 0,Y 406.281,Z 340.946,A -85,B 0,C 180,E1 -10869.792,E2 -10869.792} C_VEL
LIN {X 0,Y 410.634,Z 365.574,A -85,B 0,C 180,E1 -10870.504,E2 -10870.504} C_VEL
LIN {X 0,Y 411.253,Z 372.297,A -85,B 0,C 180,E1 -10870.664,E2 -10870.664} C_VEL
LIN {X 0,Y 410.143,Z 450.003,A -85,B 0,C 180,E1 -10872.067,E2 -10872.067} C_VEL
LIN {X 0,Y 409.416,Z 463.775,A -85,B 0,C 180,E1 -10872.518,E2 -10872.518} C_VEL
LIN {X 0,Y 408.723,Z 476.128,A -85,B 0,C 180,E1 -10873.132,E2 -10873.132} C_VEL
LIN {X 0,Y 407.733,Z 488.764,A -85,B 0,C 180,E1 -10873.991,E2 -10873.991} C_VEL
LIN {X 0,Y 406.793,Z 500.011,A -85,B 0,C 180,E1 -10874.98,E2 -10874.98} C_VEL
LIN {X 0,Y 405.909,Z 510.176,A -85,B 0,C 180,E1 -10876.099,E2 -10876.099} C_VEL
LIN {X 0,Y 405.093,Z 520.15,A -85,B 0,C 180,E1 -10877.475,E2 -10877.475} C_VEL
LIN {X 0,Y 404.166,Z 528.954,A -85,B 0,C 180,E1 -10878.972,E2 -10878.972} C_VEL
LIN {X 0,Y 403.626,Z 536.024,A -85,B 0,C 180,E1 -10880.478,E2 -10880.478} C_VEL
LIN {X 0,Y 403.249,Z 541.687,A -85,B 0,C 180,E1 -10881.985,E2 -10881.985} C_VEL
LIN {X 0,Y 402.938,Z 546.989,A -85,B 0,C 180,E1 -10883.822,E2 -10883.822} C_VEL
LIN {X 0,Y 402.931,Z 549.571,A -85,B 0,C 180,E1 -10884.997,E2 -10884.997} C_VEL
LIN {X 0,Y 402.827,Z 552.568,A -85,B 0,C 180,E1 -10886.999,E2 -10886.999} C_VEL
LIN {X 0,Y 402.907,Z 553.477,A -85,B 0,C 180,E1 -10888,E2 -10888} C_VEL
LIN {X 0,Y 402.866,Z 553.958,A -85,B 0,C 180,E1 -10889,E2 -10889} C_VEL
LIN {X 0,Y 402.871,Z 554.03,A -85,B 0,C 180,E1 -10890,E2 -10890} C_VEL
LIN {X 0,Y 402.912,Z 553.016,A -85,B 0,C 180,E1 -10891.999,E2 -10891.999} C_VEL
LIN {X 0,Y 402.859,Z 551.888,A -85,B 0,C 180,E1 -10893,E2 -10893} C_VEL
LIN {X 0,Y 402.858,Z 550.321,A -85,B 0,C 180,E1 -10894.001,E2 -10894.001} C_VEL
LIN {X 0,Y 402.912,Z 547.169,A -85,B 0,C 180,E1 -10895.505,E2 -10895.505} C_VEL
LIN {X 0,Y 403.075,Z 542.943,A -85,B 0,C 180,E1 -10897.01,E2 -10897.01} C_VEL
LIN {X 0,Y 403.363,Z 536.503,A -85,B 0,C 180,E1 -10898.769,E2 -10898.769} C_VEL
LIN {X 0,Y 403.761,Z 529.467,A -85,B 0,C 180,E1 -10900.277,E2 -10900.277} C_VEL
LIN {X 0,Y 404.387,Z 520.641,A -85,B 0,C 180,E1 -10901.783,E2 -10901.783} C_VEL
LIN {X 0,Y 405.054,Z 511.594,A -85,B 0,C 180,E1 -10903.035,E2 -10903.035} C_VEL
LIN {X 0,Y 405.735,Z 501.632,A -85,B 0,C 180,E1 -10904.162,E2 -10904.162} C_VEL
LIN {X 0,Y 406.475,Z 490.583,A -85,B 0,C 180,E1 -10905.159,E2 -10905.159} C_VEL
LIN {X 0,Y 407.255,Z 478.186,A -85,B 0,C 180,E1 -10906.028,E2 -10906.028} C_VEL
LIN {X 0,Y 407.855,Z 466.436,A -85,B 0,C 180,E1 -10906.647,E2 -10906.647} C_VEL
LIN {X 0,Y 408.388,Z 453.862,A -85,B 0,C 180,E1 -10907.107,E2 -10907.107} C_VEL
LIN {X 0,Y 408.743,Z 437.812,A -85,B 0,C 180,E1 -10907.446,E2 -10907.446} C_VEL
LIN {X 0,Y 409.301,Z 367.933,A -85,B 0,C 180,E1 -10908.676,E2 -10908.676} C_VEL
LIN {X 0,Y 405.434,Z 341.207,A -85,B 0,C 180,E1 -10909.319,E2 -10909.319} C_VEL
LIN {X 0,Y 406.472,Z 324.437,A -85,B 0,C 180,E1 -10912.625,E2 -10912.625} C_VEL
LIN {X 0,Y 407.036,Z 315.113,A -85,B 0,C 180,E1 -10914.48,E2 -10914.48} C_VEL
LIN {X 0,Y 405.058,Z 304.204,A -85,B 0,C 180,E1 -10916.815,E2 -10916.815} C_VEL
LIN {X 0,Y 404.268,Z 300.13,A -85,B 0,C 180,E1 -10917.721,E2 -10917.721} C_VEL
LIN {X 0,Y 404.139,Z 300.14,A -85,B 0,C 180,E1 -10921.557,E2 -10921.557} C_VEL
LIN {X 0,Y 404.184,Z 300.134,A -85,B 0,C 180,E1 -10925.015,E2 -10925.015} C_VEL
LIN {X 0,Y 404.149,Z 300.14,A -85,B 0,C 180,E1 -10928.757,E2 -10928.757} C_VEL
LIN {X 0,Y 404.121,Z 300.142,A -85,B 0,C 180,E1 -10931.599,E2 -10931.599} C_VEL
LIN {X 0,Y 404.143,Z 300.146,A -85,B 0,C 180,E1 -10934.521,E2 -10934.521} C_VEL
LIN {X 0,Y 404.134,Z 300.14,A -85,B 0,C 180,E1 -10937.295,E2 -10937.295} C_VEL
LIN {X 0,Y 404.166,Z 300.136,A -85,B 0,C 180,E1 -10939.955,E2 -10939.955} C_VEL
LIN {X 0,Y 404.134,Z 300.143,A -85,B 0,C 180,E1 -10943.124,E2 -10943.124} C_VEL
LIN {X 0,Y 404.142,Z 300.14,A -85,B 0,C 180,E1 -10946.187,E2 -10946.187} C_VEL
LIN {X 0,Y 404.142,Z 300.139,A -85,B 0,C 180,E1 -10949.714,E2 -10949.714} C_VEL
LIN {X 0,Y 404.192,Z 300.139,A -85,B 0,C 180,E1 -10953.122,E2 -10953.122} C_VEL
LIN {X 0,Y 404.173,Z 300.139,A -85,B 0,C 180,E1 -10955.334,E2 -10955.334} C_VEL
LIN {X 0,Y 404.134,Z 300.141,A -85,B 0,C 180,E1 -10958.58,E2 -10958.58} C_VEL
LIN {X 0,Y 404.206,Z 300.132,A -85,B 0,C 180,E1 -10961.762,E2 -10961.762} C_VEL
LIN {X 0,Y 404.202,Z 300.134,A -85,B 0,C 180,E1 -10964.882,E2 -10964.882} C_VEL
LIN {X 0,Y 404.252,Z 300.126,A -85,B 0,C 180,E1 -10967.958,E2 -10967.958} C_VEL
LIN {X 0,Y 404.4,Z 300.108,A -85,B 0,C 180,E1 -10972.128,E2 -10972.128} C_VEL
LIN {X 0,Y 404.417,Z 300.107,A -85,B 0,C 180,E1 -10974.015,E2 -10974.015} C_VEL
LIN {X 0,Y 404.474,Z 300.101,A -85,B 0,C 180,E1 -10978.008,E2 -10978.008} C_VEL
LIN {X 0,Y 404.604,Z 300.085,A -85,B 0,C 180,E1 -10980,E2 -10980} C_VEL
LIN {X 0,Y 404.412,Z 300.105,A -85,B 0,C 180,E1 -10982.988,E2 -10982.988} C_VEL
LIN {X 0,Y 404.366,Z 300.112,A -85,B 0,C 180,E1 -10986.513,E2 -10986.513} C_VEL
LIN {X 0,Y 404.283,Z 300.121,A -85,B 0,C 180,E1 -10989.001,E2 -10989.001} C_VEL
LIN {X 0,Y 404.251,Z 300.133,A -85,B 0,C 180,E1 -10992.041,E2 -10992.041} C_VEL
LIN {X 0,Y 404.2,Z 300.131,A -85,B 0,C 180,E1 -10995.118,E2 -10995.118} C_VEL
LIN {X 0,Y 404.203,Z 300.139,A -85,B 0,C 180,E1 -10998.238,E2 -10998.238} C_VEL
LIN {X 0,Y 404.132,Z 300.14,A -85,B 0,C 180,E1 -11001.42,E2 -11001.42} C_VEL
LIN {X 0,Y 404.165,Z 300.14,A -85,B 0,C 180,E1 -11004.666,E2 -11004.666} C_VEL
LIN {X 0,Y 404.19,Z 300.135,A -85,B 0,C 180,E1 -11008,E2 -11008} C_VEL
LIN {X 0,Y 404.134,Z 300.14,A -85,B 0,C 180,E1 -11011.558,E2 -11011.558} C_VEL
LIN {X 0,Y 404.179,Z 300.138,A -85,B 0,C 180,E1 -11015.016,E2 -11015.016} C_VEL
LIN {X 0,Y 404.146,Z 300.146,A -85,B 0,C 180,E1 -11018.758,E2 -11018.758} C_VEL
LIN {X 0,Y 404.118,Z 300.142,A -85,B 0,C 180,E1 -11021.6,E2 -11021.6} C_VEL
LIN {X 0,Y 404.141,Z 300.141,A -85,B 0,C 180,E1 -11024.522,E2 -11024.522} C_VEL
LIN {X 0,Y 404.12,Z 300.146,A -85,B 0,C 180,E1 -11027.294,E2 -11027.294} C_VEL
LIN {X 0,Y 404.128,Z 300.141,A -85,B 0,C 180,E1 -11029.951,E2 -11029.951} C_VEL
LIN {X 0,Y 404.131,Z 300.147,A -85,B 0,C 180,E1 -11033.126,E2 -11033.126} C_VEL
LIN {X 0,Y 404.141,Z 300.139,A -85,B 0,C 180,E1 -11036.188,E2 -11036.188} C_VEL
LIN {X 0,Y 404.141,Z 300.142,A -85,B 0,C 180,E1 -11039.715,E2 -11039.715} C_VEL
LIN {X 0,Y 404.103,Z 300.147,A -85,B 0,C 180,E1 -11043.117,E2 -11043.117} C_VEL
LIN {X 0,Y 404.146,Z 300.138,A -85,B 0,C 180,E1 -11046.425,E2 -11046.425} C_VEL
LIN {X 0,Y 404.189,Z 300.137,A -85,B 0,C 180,E1 -11049.875,E2 -11049.875} C_VEL
LIN {X 0,Y 404.214,Z 300.13,A -85,B 0,C 180,E1 -11052.994,E2 -11052.994} C_VEL
LIN {X 0,Y 404.282,Z 300.125,A -85,B 0,C 180,E1 -11056.939,E2 -11056.939} C_VEL
LIN {X 0,Y 404.323,Z 300.28,A -85,B 0,C 180,E1 -11057.834,E2 -11057.834} C_VEL
LIN {X 0,Y 405.897,Z 309.659,A -85,B 0,C 180,E1 -11060.03,E2 -11060.03} C_VEL
LIN {X 0,Y 405.881,Z 312.977,A -85,B 0,C 180,E1 -11060.767,E2 -11060.767} C_VEL
LIN {X 0,Y 409.742,Z 333.765,A -85,B 0,C 180,E1 -11061.312,E2 -11061.312} C_VEL
LIN {X 0,Y 408.653,Z 421.174,A -85,B 0,C 180,E1 -11062.869,E2 -11062.869} C_VEL
LIN {X 0,Y 408.245,Z 434.798,A -85,B 0,C 180,E1 -11063.327,E2 -11063.327} C_VEL
LIN {X 0,Y 407.829,Z 447.033,A -85,B 0,C 180,E1 -11063.942,E2 -11063.942} C_VEL
LIN {X 0,Y 407.167,Z 459.596,A -85,B 0,C 180,E1 -11064.801,E2 -11064.801} C_VEL
LIN {X 0,Y 406.242,Z 470.82,A -85,B 0,C 180,E1 -11065.784,E2 -11065.784} C_VEL
LIN {X 0,Y 405.515,Z 480.9,A -85,B 0,C 180,E1 -11066.896,E2 -11066.896} C_VEL
LIN {X 0,Y 404.919,Z 490.764,A -85,B 0,C 180,E1 -11068.26,E2 -11068.26} C_VEL
LIN {X 0,Y 404.583,Z 495.318,A -85,B 0,C 180,E1 -11068.998,E2 -11068.998} C_VEL
LIN {X 0,Y 403.695,Z 499.025,A -85,B 0,C 180,E1 -11069.639,E2 -11069.639} C_VEL
LIN {X 0,Y 400.458,Z 504.635,A -85,B 0,C 180,E1 -11070.71,E2 -11070.71} C_VEL
LIN {X 0,Y 397.229,Z 509.55,A -85,B 0,C 180,E1 -11071.861,E2 -11071.861} C_VEL
LIN {X 0,Y 396.37,Z 512.167,A -85,B 0,C 180,E1 -11072.618,E2 -11072.618} C_VEL
LIN {X 0,Y 396.042,Z 516.419,A -85,B 0,C 180,E1 -11074.071,E2 -11074.071} C_VEL
LIN {X 0,Y 396.03,Z 518.78,A -85,B 0,C 180,E1 -11075.091,E2 -11075.091} C_VEL
LIN {X 0,Y 395.991,Z 521.118,A -85,B 0,C 180,E1 -11076.343,E2 -11076.343} C_VEL
LIN {X 0,Y 395.75,Z 523.338,A -85,B 0,C 180,E1 -11078.168,E2 -11078.168} C_VEL
LIN {X 0,Y 395.678,Z 524.315,A -85,B 0,C 180,E1 -11080.231,E2 -11080.231} C_VEL
LIN {X 0,Y 395.749,Z 524.211,A -85,B 0,C 180,E1 -11081.265,E2 -11081.265} C_VEL
LIN {X 0,Y 395.84,Z 523.553,A -85,B 0,C 180,E1 -11082.445,E2 -11082.445} C_VEL
LIN {X 0,Y 395.952,Z 521.37,A -85,B 0,C 180,E1 -11084.389,E2 -11084.389} C_VEL
LIN {X 0,Y 396.256,Z 518.484,A -85,B 0,C 180,E1 -11085.957,E2 -11085.957} C_VEL
LIN {X 0,Y 396.574,Z 514.52,A -85,B 0,C 180,E1 -11087.534,E2 -11087.534} C_VEL
LIN {X 0,Y 397.195,Z 508.337,A -85,B 0,C 180,E1 -11089.376,E2 -11089.376} C_VEL
LIN {X 0,Y 397.867,Z 501.505,A -85,B 0,C 180,E1 -11090.959,E2 -11090.959} C_VEL
LIN {X 0,Y 398.707,Z 492.943,A -85,B 0,C 180,E1 -11092.544,E2 -11092.544} C_VEL
LIN {X 0,Y 399.644,Z 483.931,A -85,B 0,C 180,E1 -11093.872,E2 -11093.872} C_VEL
LIN {X 0,Y 400.656,Z 472.978,A -85,B 0,C 180,E1 -11095.175,E2 -11095.175} C_VEL
LIN {X 0,Y 401.639,Z 461.837,A -85,B 0,C 180,E1 -11096.217,E2 -11096.217} C_VEL
LIN {X 0,Y 402.491,Z 449.109,A -85,B 0,C 180,E1 -11097.14,E2 -11097.14} C_VEL
LIN {X 0,Y 403.143,Z 436.937,A -85,B 0,C 180,E1 -11097.796,E2 -11097.796} C_VEL
LIN {X 0,Y 403.431,Z 424.411,A -85,B 0,C 180,E1 -11098.27,E2 -11098.27} C_VEL
LIN {X 0,Y 403.896,Z 409.363,A -85,B 0,C 180,E1 -11098.588,E2 -11098.588} C_VEL
LIN {X 0,Y 405.134,Z 335.598,A -85,B 0,C 180,E1 -11099.908,E2 -11099.908} C_VEL
LIN {X 0,Y 400.651,Z 316.325,A -85,B 0,C 180,E1 -11100.551,E2 -11100.551} C_VEL
LIN {X 0,Y 399.714,Z 313.365,A -85,B 0,C 180,E1 -11100.684,E2 -11100.684} C_VEL
LIN {X 0,Y 397.587,Z 303.13,A -85,B 0,C 180,E1 -11103.228,E2 -11103.228} C_VEL
LIN {X 0,Y 397.106,Z 301.022,A -85,B 0,C 180,E1 -11103.785,E2 -11103.785} C_VEL
LIN {X 0,Y 397.093,Z 301.013,A -85,B 0,C 180,E1 -11107.209,E2 -11107.209} C_VEL
LIN {X 0,Y 397.101,Z 301.021,A -85,B 0,C 180,E1 -11110.446,E2 -11110.446} C_VEL
LIN {X 0,Y 397.1,Z 301.019,A -85,B 0,C 180,E1 -11113.649,E2 -11113.649} C_VEL
LIN {X 0,Y 397.101,Z 301.022,A -85,B 0,C 180,E1 -11116.521,E2 -11116.521} C_VEL
LIN {X 0,Y 397.113,Z 301.018,A -85,B 0,C 180,E1 -11120.423,E2 -11120.423} C_VEL
LIN {X 0,Y 397.107,Z 301.014,A -85,B 0,C 180,E1 -11124.265,E2 -11124.265} C_VEL
LIN {X 0,Y 397.114,Z 301.015,A -85,B 0,C 180,E1 -11126.727,E2 -11126.727} C_VEL
LIN {X 0,Y 397.124,Z 301.009,A -85,B 0,C 180,E1 -11130.296,E2 -11130.296} C_VEL
LIN {X 0,Y 397.193,Z 301,A -85,B 0,C 180,E1 -11132.61,E2 -11132.61} C_VEL
LIN {X 0,Y 397.128,Z 301.006,A -85,B 0,C 180,E1 -11135.982,E2 -11135.982} C_VEL
LIN {X 0,Y 397.138,Z 301.009,A -85,B 0,C 180,E1 -11139.705,E2 -11139.705} C_VEL
LIN {X 0,Y 397.181,Z 301.008,A -85,B 0,C 180,E1 -11142.845,E2 -11142.845} C_VEL
LIN {X 0,Y 397.228,Z 301.001,A -85,B 0,C 180,E1 -11146.703,E2 -11146.703} C_VEL
LIN {X 0,Y 397.217,Z 301.004,A -85,B 0,C 180,E1 -11149.809,E2 -11149.809} C_VEL
LIN {X 0,Y 397.362,Z 300.981,A -85,B 0,C 180,E1 -11152.888,E2 -11152.888} C_VEL
LIN {X 0,Y 397.253,Z 300.996,A -85,B 0,C 180,E1 -11154.925,E2 -11154.925} C_VEL
LIN {X 0,Y 397.449,Z 300.972,A -85,B 0,C 180,E1 -11157.973,E2 -11157.973} C_VEL
LIN {X 0,Y 397.578,Z 300.961,A -85,B 0,C 180,E1 -11160,E2 -11160} C_VEL
LIN {X 0,Y 397.375,Z 300.977,A -85,B 0,C 180,E1 -11163.042,E2 -11163.042} C_VEL
LIN {X 0,Y 397.362,Z 300.976,A -85,B 0,C 180,E1 -11167.112,E2 -11167.112} C_VEL
LIN {X 0,Y 397.218,Z 301.006,A -85,B 0,C 180,E1 -11170.191,E2 -11170.191} C_VEL
LIN {X 0,Y 397.227,Z 301,A -85,B 0,C 180,E1 -11173.321,E2 -11173.321} C_VEL
LIN {X 0,Y 397.182,Z 301.006,A -85,B 0,C 180,E1 -11177.155,E2 -11177.155} C_VEL
LIN {X 0,Y 397.103,Z 301.016,A -85,B 0,C 180,E1 -11180.73,E2 -11180.73} C_VEL
LIN {X 0,Y 397.129,Z 301.012,A -85,B 0,C 180,E1 -11184.019,E2 -11184.019} C_VEL
LIN {X 0,Y 397.195,Z 301.005,A -85,B 0,C 180,E1 -11187.39,E2 -11187.39} C_VEL
LIN {X 0,Y 397.08,Z 301.026,A -85,B 0,C 180,E1 -11190.883,E2 -11190.883} C_VEL
LIN {X 0,Y 397.126,Z 301.015,A -85,B 0,C 180,E1 -11194.494,E2 -11194.494} C_VEL
LIN {X 0,Y 397.102,Z 301.016,A -85,B 0,C 180,E1 -11198.275,E2 -11198.275} C_VEL
LIN {X 0,Y 397.09,Z 301.005,A -85,B 0,C 180,E1 -11200.909,E2 -11200.909} C_VEL
LIN {X 0,Y 397.102,Z 301.019,A -85,B 0,C 180,E1 -11203.649,E2 -11203.649} C_VEL
LIN {X 0,Y 397.103,Z 301.017,A -85,B 0,C 180,E1 -11206.521,E2 -11206.521} C_VEL
LIN {X 0,Y 397.114,Z 301.016,A -85,B 0,C 180,E1 -11210.423,E2 -11210.423} C_VEL
LIN {X 0,Y 397.11,Z 301.019,A -85,B 0,C 180,E1 -11214.265,E2 -11214.265} C_VEL
LIN {X 0,Y 397.117,Z 301.019,A -85,B 0,C 180,E1 -11216.727,E2 -11216.727} C_VEL
LIN {X 0,Y 397.172,Z 301.077,A -85,B 0,C 180,E1 -11220.7,E2 -11220.7} C_VEL
LIN {X 0,Y 399.969,Z 313.486,A -85,B 0,C 180,E1 -11223.656,E2 -11223.656} C_VEL
LIN {X 0,Y 401.058,Z 319.978,A -85,B 0,C 180,E1 -11225.129,E2 -11225.129} C_VEL
LIN {X 0,Y 399.643,Z 337.563,A -85,B 0,C 180,E1 -11228.756,E2 -11228.756} C_VEL
LIN {X 0,Y 399.414,Z 340.552,A -85,B 0,C 180,E1 -11229.366,E2 -11229.366} C_VEL
LIN {X 0,Y 404.006,Z 365.894,A -85,B 0,C 180,E1 -11230.13,E2 -11230.13} C_VEL
LIN {X 0,Y 404.673,Z 373.038,A -85,B 0,C 180,E1 -11230.303,E2 -11230.303} C_VEL
LIN {X 0,Y 403.513,Z 449.337,A -85,B 0,C 180,E1 -11231.7,E2 -11231.7} C_VEL
LIN {X 0,Y 402.832,Z 462.396,A -85,B 0,C 180,E1 -11232.124,E2 -11232.124} C_VEL
LIN {X 0,Y 402.05,Z 475.605,A -85,B 0,C 180,E1 -11232.778,E2 -11232.778} C_VEL
LIN {X 0,Y 401.079,Z 487.519,A -85,B 0,C 180,E1 -11233.587,E2 -11233.587} C_VEL
LIN {X 0,Y 400.04,Z 498.945,A -85,B 0,C 180,E1 -11234.59,E2 -11234.59} C_VEL
LIN {X 0,Y 399.076,Z 509.263,A -85,B 0,C 180,E1 -11235.726,E2 -11235.726} C_VEL
LIN {X 0,Y 398.274,Z 518.558,A -85,B 0,C 180,E1 -11236.998,E2 -11236.998} C_VEL
LIN {X 0,Y 397.351,Z 527.58,A -85,B 0,C 180,E1 -11238.522,E2 -11238.522} C_VEL
LIN {X 0,Y 396.692,Z 534.869,A -85,B 0,C 180,E1 -11240.053,E2 -11240.053} C_VEL
LIN {X 0,Y 396.197,Z 541.566,A -85,B 0,C 180,E1 -11241.841,E2 -11241.841} C_VEL
LIN {X 0,Y 395.921,Z 546.008,A -85,B 0,C 180,E1 -11243.375,E2 -11243.375} C_VEL
LIN {X 0,Y 395.843,Z 549.384,A -85,B 0,C 180,E1 -11244.907,E2 -11244.907} C_VEL
LIN {X 0,Y 395.776,Z 551.068,A -85,B 0,C 180,E1 -11245.927,E2 -11245.927} C_VEL
LIN {X 0,Y 395.804,Z 553.244,A -85,B 0,C 180,E1 -11247.965,E2 -11247.965} C_VEL
LIN {X 0,Y 395.795,Z 553.701,A -85,B 0,C 180,E1 -11248.982,E2 -11248.982} C_VEL
LIN {X 0,Y 395.797,Z 553.759,A -85,B 0,C 180,E1 -11250,E2 -11250} C_VEL
LIN {X 0,Y 395.81,Z 553.432,A -85,B 0,C 180,E1 -11251.017,E2 -11251.017} C_VEL
LIN {X 0,Y 395.825,Z 552.716,A -85,B 0,C 180,E1 -11252.035,E2 -11252.035} C_VEL
LIN {X 0,Y 395.76,Z 551.56,A -85,B 0,C 180,E1 -11253.053,E2 -11253.053} C_VEL
LIN {X 0,Y 395.821,Z 549.055,A -85,B 0,C 180,E1 -11254.582,E2 -11254.582} C_VEL
LIN {X 0,Y 395.929,Z 544.229,A -85,B 0,C 180,E1 -11256.574,E2 -11256.574} C_VEL
LIN {X 0,Y 396.134,Z 539.048,A -85,B 0,C 180,E1 -11258.159,E2 -11258.159} C_VEL
LIN {X 0,Y 396.505,Z 532.711,A -85,B 0,C 180,E1 -11259.694,E2 -11259.694} C_VEL
LIN {X 0,Y 397.021,Z 524.758,A -85,B 0,C 180,E1 -11261.228,E2 -11261.228} C_VEL
LIN {X 0,Y 397.701,Z 516.653,A -85,B 0,C 180,E1 -11262.502,E2 -11262.502} C_VEL
LIN {X 0,Y 398.411,Z 506.928,A -85,B 0,C 180,E1 -11263.755,E2 -11263.755} C_VEL
LIN {X 0,Y 399.048,Z 497.013,A -85,B 0,C 180,E1 -11264.795,E2 -11264.795} C_VEL
LIN {X 0,Y 399.783,Z 486.528,A -85,B 0,C 180,E1 -11265.681,E2 -11265.681} C_VEL
LIN {X 0,Y 400.579,Z 473.905,A -85,B 0,C 180,E1 -11266.499,E2 -11266.499} C_VEL
LIN {X 0,Y 401.227,Z 460.555,A -85,B 0,C 180,E1 -11267.127,E2 -11267.127} C_VEL
LIN {X 0,Y 401.725,Z 448.334,A -85,B 0,C 180,E1 -11267.498,E2 -11267.498} C_VEL
LIN {X 0,Y 402.534,Z 369.173,A -85,B 0,C 180,E1 -11268.925,E2 -11268.925} C_VEL
LIN {X 0,Y 398.509,Z 340.808,A -85,B 0,C 180,E1 -11269.644,E2 -11269.644} C_VEL
LIN {X 0,Y 399.62,Z 323.903,A -85,B 0,C 180,E1 -11273.035,E2 -11273.035} C_VEL
LIN {X 0,Y 400.017,Z 315.901,A -85,B 0,C 180,E1 -11274.661,E2 -11274.661} C_VEL
LIN {X 0,Y 398.013,Z 304.977,A -85,B 0,C 180,E1 -11277.044,E2 -11277.044} C_VEL
LIN {X 0,Y 397.208,Z 301.01,A -85,B 0,C 180,E1 -11277.956,E2 -11277.956} C_VEL
LIN {X 0,Y 397.082,Z 301.022,A -85,B 0,C 180,E1 -11281.836,E2 -11281.836} C_VEL
LIN {X 0,Y 397.125,Z 301.017,A -85,B 0,C 180,E1 -11284.493,E2 -11284.493} C_VEL
LIN {X 0,Y 397.099,Z 301.023,A -85,B 0,C 180,E1 -11288.275,E2 -11288.275} C_VEL
LIN {X 0,Y 397.087,Z 301.019,A -85,B 0,C 180,E1 -11290.908,E2 -11290.908} C_VEL
LIN {X 0,Y 397.099,Z 301.016,A -85,B 0,C 180,E1 -11293.648,E2 -11293.648} C_VEL
LIN {X 0,Y 397.1,Z 301.024,A -85,B 0,C 180,E1 -11296.52,E2 -11296.52} C_VEL
LIN {X 0,Y 397.111,Z 301.019,A -85,B 0,C 180,E1 -11300.422,E2 -11300.422} C_VEL
LIN {X 0,Y 397.105,Z 301.017,A -85,B 0,C 180,E1 -11304.265,E2 -11304.265} C_VEL
LIN {X 0,Y 397.111,Z 301.021,A -85,B 0,C 180,E1 -11306.726,E2 -11306.726} C_VEL
LIN {X 0,Y 397.121,Z 301.014,A -85,B 0,C 180,E1 -11310.295,E2 -11310.295} C_VEL
LIN {X 0,Y 397.191,Z 301.008,A -85,B 0,C 180,E1 -11312.609,E2 -11312.609} C_VEL
LIN {X 0,Y 397.129,Z 301.012,A -85,B 0,C 180,E1 -11315.981,E2 -11315.981} C_VEL
LIN {X 0,Y 397.134,Z 301.013,A -85,B 0,C 180,E1 -11319.704,E2 -11319.704} C_VEL
LIN {X 0,Y 397.177,Z 301.009,A -85,B 0,C 180,E1 -11322.844,E2 -11322.844} C_VEL
LIN {X 0,Y 397.224,Z 301.001,A -85,B 0,C 180,E1 -11326.702,E2 -11326.702} C_VEL
LIN {X 0,Y 397.213,Z 301.005,A -85,B 0,C 180,E1 -11329.809,E2 -11329.809} C_VEL
LIN {X 0,Y 397.347,Z 300.986,A -85,B 0,C 180,E1 -11332.888,E2 -11332.888} C_VEL
LIN {X 0,Y 397.248,Z 300.998,A -85,B 0,C 180,E1 -11334.925,E2 -11334.925} C_VEL
LIN {X 0,Y 397.443,Z 300.977,A -85,B 0,C 180,E1 -11337.973,E2 -11337.973} C_VEL
LIN {X 0,Y 397.573,Z 300.961,A -85,B 0,C 180,E1 -11340,E2 -11340} C_VEL
LIN {X 0,Y 397.371,Z 300.983,A -85,B 0,C 180,E1 -11343.041,E2 -11343.041} C_VEL
LIN {X 0,Y 397.32,Z 300.99,A -85,B 0,C 180,E1 -11346.506,E2 -11346.506} C_VEL
LIN {X 0,Y 397.246,Z 300.998,A -85,B 0,C 180,E1 -11349.162,E2 -11349.162} C_VEL
LIN {X 0,Y 397.214,Z 301.007,A -85,B 0,C 180,E1 -11352.258,E2 -11352.258} C_VEL
LIN {X 0,Y 397.173,Z 301.007,A -85,B 0,C 180,E1 -11355.392,E2 -11355.392} C_VEL
LIN {X 0,Y 397.155,Z 301.012,A -85,B 0,C 180,E1 -11358.574,E2 -11358.574} C_VEL
LIN {X 0,Y 397.09,Z 301.019,A -85,B 0,C 180,E1 -11361.819,E2 -11361.819} C_VEL
LIN {X 0,Y 397.145,Z 301.01,A -85,B 0,C 180,E1 -11365.512,E2 -11365.512} C_VEL
LIN {X 0,Y 397.117,Z 301.021,A -85,B 0,C 180,E1 -11368.544,E2 -11368.544} C_VEL
LIN {X 0,Y 397.073,Z 301.021,A -85,B 0,C 180,E1 -11372.072,E2 -11372.072} C_VEL
LIN {X 0,Y 397.114,Z 301.014,A -85,B 0,C 180,E1 -11375.504,E2 -11375.504} C_VEL
LIN {X 0,Y 397.122,Z 301.02,A -85,B 0,C 180,E1 -11378.861,E2 -11378.861} C_VEL
LIN {X 0,Y 397.064,Z 301.022,A -85,B 0,C 180,E1 -11382.268,E2 -11382.268} C_VEL
LIN {X 0,Y 397.082,Z 301.024,A -85,B 0,C 180,E1 -11385.069,E2 -11385.069} C_VEL
LIN {X 0,Y 397.05,Z 301.022,A -85,B 0,C 180,E1 -11388.024,E2 -11388.024} C_VEL
LIN {X 0,Y 397.09,Z 301.019,A -85,B 0,C 180,E1 -11391.724,E2 -11391.724} C_VEL
LIN {X 0,Y 397.121,Z 301.018,A -85,B 0,C 180,E1 -11395.507,E2 -11395.507} C_VEL
LIN {X 0,Y 397.075,Z 301.024,A -85,B 0,C 180,E1 -11399.118,E2 -11399.118} C_VEL
LIN {X 0,Y 397.06,Z 301.021,A -85,B 0,C 180,E1 -11402.252,E2 -11402.252} C_VEL
LIN {X 0,Y 397.1,Z 301.017,A -85,B 0,C 180,E1 -11404.865,E2 -11404.865} C_VEL
LIN {X 0,Y 397.093,Z 301.018,A -85,B 0,C 180,E1 -11408.182,E2 -11408.182} C_VEL
LIN {X 0,Y 397.155,Z 301.014,A -85,B 0,C 180,E1 -11411.427,E2 -11411.427} C_VEL
LIN {X 0,Y 397.177,Z 301.009,A -85,B 0,C 180,E1 -11414.608,E2 -11414.608} C_VEL
LIN {X 0,Y 397.277,Z 301.121,A -85,B 0,C 180,E1 -11417.619,E2 -11417.619} C_VEL
LIN {X 0,Y 398.889,Z 310.496,A -85,B 0,C 180,E1 -11419.853,E2 -11419.853} C_VEL
LIN {X 0,Y 398.955,Z 313.211,A -85,B 0,C 180,E1 -11420.47,E2 -11420.47} C_VEL
LIN {X 0,Y 402.95,Z 335.077,A -85,B 0,C 180,E1 -11421.054,E2 -11421.054} C_VEL
LIN {X 0,Y 401.824,Z 420.453,A -85,B 0,C 180,E1 -11422.589,E2 -11422.589} C_VEL
LIN {X 0,Y 401.433,Z 433.651,A -85,B 0,C 180,E1 -11423.024,E2 -11423.024} C_VEL
LIN {X 0,Y 400.955,Z 446.287,A -85,B 0,C 180,E1 -11423.648,E2 -11423.648} C_VEL
LIN {X 0,Y 400.343,Z 458.349,A -85,B 0,C 180,E1 -11424.46,E2 -11424.46} C_VEL
LIN {X 0,Y 399.612,Z 467.267,A -85,B 0,C 180,E1 -11425.208,E2 -11425.208} C_VEL
LIN {X 0,Y 398.849,Z 478.036,A -85,B 0,C 180,E1 -11426.338,E2 -11426.338} C_VEL
LIN {X 0,Y 398.142,Z 486.841,A -85,B 0,C 180,E1 -11427.471,E2 -11427.471} C_VEL
LIN {X 0,Y 397.523,Z 496.389,A -85,B 0,C 180,E1 -11428.987,E2 -11428.987} C_VEL
LIN {X 0,Y 396.856,Z 504.024,A -85,B 0,C 180,E1 -11430.508,E2 -11430.508} C_VEL
LIN {X 0,Y 396.464,Z 510.148,A -85,B 0,C 180,E1 -11432.032,E2 -11432.032} C_VEL
LIN {X 0,Y 396.37,Z 512.167,A -85,B 0,C 180,E1 -11432.618,E2 -11432.618} C_VEL
LIN {X 0,Y 395.566,Z 514.595,A -85,B 0,C 180,E1 -11433.392,E2 -11433.392} C_VEL
LIN {X 0,Y 392.575,Z 518.062,A -85,B 0,C 180,E1 -11434.671,E2 -11434.671} C_VEL
LIN {X 0,Y 390.075,Z 520.313,A -85,B 0,C 180,E1 -11435.728,E2 -11435.728} C_VEL
LIN {X 0,Y 388.947,Z 521.717,A -85,B 0,C 180,E1 -11436.56,E2 -11436.56} C_VEL
LIN {X 0,Y 388.823,Z 522.096,A -85,B 0,C 180,E1 -11436.845,E2 -11436.845} C_VEL
LIN {X 0,Y 388.648,Z 523.708,A -85,B 0,C 180,E1 -11438.318,E2 -11438.318} C_VEL
LIN {X 0,Y 388.61,Z 524.601,A -85,B 0,C 180,E1 -11440.42,E2 -11440.42} C_VEL
LIN {X 0,Y 388.664,Z 524.418,A -85,B 0,C 180,E1 -11441.473,E2 -11441.473} C_VEL
LIN {X 0,Y 388.769,Z 523.825,A -85,B 0,C 180,E1 -11442.529,E2 -11442.529} C_VEL
LIN {X 0,Y 388.781,Z 522.839,A -85,B 0,C 180,E1 -11443.592,E2 -11443.592} C_VEL
LIN {X 0,Y 388.92,Z 521.437,A -85,B 0,C 180,E1 -11444.655,E2 -11444.655} C_VEL
LIN {X 0,Y 389.247,Z 518.466,A -85,B 0,C 180,E1 -11446.252,E2 -11446.252} C_VEL
LIN {X 0,Y 389.618,Z 514.4,A -85,B 0,C 180,E1 -11447.858,E2 -11447.858} C_VEL
LIN {X 0,Y 390.287,Z 508.074,A -85,B 0,C 180,E1 -11449.733,E2 -11449.733} C_VEL
LIN {X 0,Y 390.982,Z 501.125,A -85,B 0,C 180,E1 -11451.346,E2 -11451.346} C_VEL
LIN {X 0,Y 391.764,Z 493.977,A -85,B 0,C 180,E1 -11452.687,E2 -11452.687} C_VEL
LIN {X 0,Y 392.71,Z 485.537,A -85,B 0,C 180,E1 -11453.989,E2 -11453.989} C_VEL
LIN {X 0,Y 393.679,Z 475.647,A -85,B 0,C 180,E1 -11455.228,E2 -11455.228} C_VEL
LIN {X 0,Y 394.672,Z 465.073,A -85,B 0,C 180,E1 -11456.293,E2 -11456.293} C_VEL
LIN {X 0,Y 395.575,Z 453.748,A -85,B 0,C 180,E1 -11457.198,E2 -11457.198} C_VEL
LIN {X 0,Y 396.298,Z 441.215,A -85,B 0,C 180,E1 -11457.96,E2 -11457.96} C_VEL
LIN {X 0,Y 396.807,Z 427.827,A -85,B 0,C 180,E1 -11458.532,E2 -11458.532} C_VEL
LIN {X 0,Y 397.177,Z 416.693,A -85,B 0,C 180,E1 -11458.828,E2 -11458.828} C_VEL
LIN {X 0,Y 398.61,Z 336.665,A -85,B 0,C 180,E1 -11460.287,E2 -11460.287} C_VEL
LIN {X 0,Y 394.25,Z 318.198,A -85,B 0,C 180,E1 -11460.924,E2 -11460.924} C_VEL
LIN {X 0,Y 392.588,Z 313.626,A -85,B 0,C 180,E1 -11461.145,E2 -11461.145} C_VEL
LIN {X 0,Y 390.078,Z 301.897,A -85,B 0,C 180,E1 -11464.179,E2 -11464.179} C_VEL
LIN {X 0,Y 390.042,Z 301.891,A -85,B 0,C 180,E1 -11467.78,E2 -11467.78} C_VEL
LIN {X 0,Y 390.056,Z 301.9,A -85,B 0,C 180,E1 -11470.821,E2 -11470.821} C_VEL
LIN {X 0,Y 390.054,Z 301.897,A -85,B 0,C 180,E1 -11473.886,E2 -11473.886} C_VEL
LIN {X 0,Y 390.056,Z 301.9,A -85,B 0,C 180,E1 -11476.79,E2 -11476.79} C_VEL
LIN {X 0,Y 390.056,Z 301.895,A -85,B 0,C 180,E1 -11479.561,E2 -11479.561} C_VEL
LIN {X 0,Y 390.043,Z 301.896,A -85,B 0,C 180,E1 -11482.449,E2 -11482.449} C_VEL
LIN {X 0,Y 390.067,Z 301.889,A -85,B 0,C 180,E1 -11486.045,E2 -11486.045} C_VEL
LIN {X 0,Y 390.046,Z 301.891,A -85,B 0,C 180,E1 -11489.869,E2 -11489.869} C_VEL
LIN {X 0,Y 390.112,Z 301.884,A -85,B 0,C 180,E1 -11493.232,E2 -11493.232} C_VEL
LIN {X 0,Y 390.076,Z 301.885,A -85,B 0,C 180,E1 -11496.761,E2 -11496.761} C_VEL
LIN {X 0,Y 390.103,Z 301.883,A -85,B 0,C 180,E1 -11499.983,E2 -11499.983} C_VEL
LIN {X 0,Y 390.137,Z 301.888,A -85,B 0,C 180,E1 -11503.248,E2 -11503.248} C_VEL
LIN {X 0,Y 390.194,Z 301.878,A -85,B 0,C 180,E1 -11506.562,E2 -11506.562} C_VEL
LIN {X 0,Y 390.204,Z 301.876,A -85,B 0,C 180,E1 -11510.671,E2 -11510.671} C_VEL
LIN {X 0,Y 390.316,Z 301.859,A -85,B 0,C 180,E1 -11512.759,E2 -11512.759} C_VEL
LIN {X 0,Y 390.225,Z 301.872,A -85,B 0,C 180,E1 -11514.834,E2 -11514.834} C_VEL
LIN {X 0,Y 390.418,Z 301.848,A -85,B 0,C 180,E1 -11517.937,E2 -11517.937} C_VEL
LIN {X 0,Y 390.548,Z 301.837,A -85,B 0,C 180,E1 -11520,E2 -11520} C_VEL
LIN {X 0,Y 390.31,Z 301.857,A -85,B 0,C 180,E1 -11523.097,E2 -11523.097} C_VEL
LIN {X 0,Y 390.327,Z 301.86,A -85,B 0,C 180,E1 -11526.202,E2 -11526.202} C_VEL
LIN {X 0,Y 390.315,Z 301.861,A -85,B 0,C 180,E1 -11528.282,E2 -11528.282} C_VEL
LIN {X 0,Y 390.171,Z 301.879,A -85,B 0,C 180,E1 -11532.483,E2 -11532.483} C_VEL
LIN {X 0,Y 390.139,Z 301.879,A -85,B 0,C 180,E1 -11535.677,E2 -11535.677} C_VEL
LIN {X 0,Y 390.106,Z 301.889,A -85,B 0,C 180,E1 -11538.922,E2 -11538.922} C_VEL
LIN {X 0,Y 390.038,Z 301.897,A -85,B 0,C 180,E1 -11542.234,E2 -11542.234} C_VEL
LIN {X 0,Y 390.12,Z 301.886,A -85,B 0,C 180,E1 -11545.744,E2 -11545.744} C_VEL
LIN {X 0,Y 390.059,Z 301.895,A -85,B 0,C 180,E1 -11549.11,E2 -11549.11} C_VEL
LIN {X 0,Y 390.044,Z 301.895,A -85,B 0,C 180,E1 -11552.722,E2 -11552.722} C_VEL
LIN {X 0,Y 390.057,Z 301.891,A -85,B 0,C 180,E1 -11555.825,E2 -11555.825} C_VEL
LIN {X 0,Y 390.069,Z 301.886,A -85,B 0,C 180,E1 -11559.218,E2 -11559.218} C_VEL
LIN {X 0,Y 390.044,Z 301.895,A -85,B 0,C 180,E1 -11562.374,E2 -11562.374} C_VEL
LIN {X 0,Y 390.045,Z 301.9,A -85,B 0,C 180,E1 -11565.355,E2 -11565.355} C_VEL
LIN {X 0,Y 390.032,Z 301.899,A -85,B 0,C 180,E1 -11568.187,E2 -11568.187} C_VEL
LIN {X 0,Y 390.089,Z 301.892,A -85,B 0,C 180,E1 -11570.907,E2 -11570.907} C_VEL
LIN {X 0,Y 390.087,Z 301.893,A -85,B 0,C 180,E1 -11574.793,E2 -11574.793} C_VEL
LIN {X 0,Y 390.026,Z 301.904,A -85,B 0,C 180,E1 -11578.496,E2 -11578.496} C_VEL
LIN {X 0,Y 390.098,Z 301.922,A -85,B 0,C 180,E1 -11580.301,E2 -11580.301} C_VEL
LIN {X 0,Y 392.748,Z 313.533,A -85,B 0,C 180,E1 -11583.139,E2 -11583.139} C_VEL
LIN {X 0,Y 394.129,Z 321.117,A -85,B 0,C 180,E1 -11584.908,E2 -11584.908} C_VEL
LIN {X 0,Y 393.08,Z 334.219,A -85,B 0,C 180,E1 -11587.67,E2 -11587.67} C_VEL
LIN {X 0,Y 392.599,Z 340.345,A -85,B 0,C 180,E1 -11588.936,E2 -11588.936} C_VEL
LIN {X 0,Y 397.229,Z 365.457,A -85,B 0,C 180,E1 -11589.716,E2 -11589.716} C_VEL
LIN {X 0,Y 398.137,Z 372.077,A -85,B 0,C 180,E1 -11589.899,E2 -11589.899} C_VEL
LIN {X 0,Y 396.913,Z 448.787,A -85,B 0,C 180,E1 -11591.322,E2 -11591.322} C_VEL
LIN {X 0,Y 396.161,Z 462.596,A -85,B 0,C 180,E1 -11591.779,E2 -11591.779} C_VEL
LIN {X 0,Y 395.395,Z 475.125,A -85,B 0,C 180,E1 -11592.412,E2 -11592.412} C_VEL
LIN {X 0,Y 394.43,Z 486.31,A -85,B 0,C 180,E1 -11593.169,E2 -11593.169} C_VEL
LIN {X 0,Y 393.339,Z 497.903,A -85,B 0,C 180,E1 -11594.188,E2 -11594.188} C_VEL
LIN {X 0,Y 392.349,Z 508.029,A -85,B 0,C 180,E1 -11595.304,E2 -11595.304} C_VEL
LIN {X 0,Y 391.513,Z 516.904,A -85,B 0,C 180,E1 -11596.505,E2 -11596.505} C_VEL
LIN {X 0,Y 390.699,Z 524.813,A -85,B 0,C 180,E1 -11597.798,E2 -11597.798} C_VEL
LIN {X 0,Y 389.916,Z 532.576,A -85,B 0,C 180,E1 -11599.353,E2 -11599.353} C_VEL
LIN {X 0,Y 389.265,Z 539.724,A -85,B 0,C 180,E1 -11601.172,E2 -11601.172} C_VEL
LIN {X 0,Y 388.939,Z 544.51,A -85,B 0,C 180,E1 -11602.733,E2 -11602.733} C_VEL
LIN {X 0,Y 388.775,Z 547.287,A -85,B 0,C 180,E1 -11603.856,E2 -11603.856} C_VEL
LIN {X 0,Y 388.7,Z 550.869,A -85,B 0,C 180,E1 -11605.852,E2 -11605.852} C_VEL
LIN {X 0,Y 388.701,Z 553.009,A -85,B 0,C 180,E1 -11607.927,E2 -11607.927} C_VEL
LIN {X 0,Y 388.726,Z 553.444,A -85,B 0,C 180,E1 -11608.964,E2 -11608.964} C_VEL
LIN {X 0,Y 388.726,Z 553.488,A -85,B 0,C 180,E1 -11610,E2 -11610} C_VEL
LIN {X 0,Y 388.741,Z 553.146,A -85,B 0,C 180,E1 -11611.036,E2 -11611.036} C_VEL
LIN {X 0,Y 388.725,Z 552.411,A -85,B 0,C 180,E1 -11612.072,E2 -11612.072} C_VEL
LIN {X 0,Y 388.664,Z 551.228,A -85,B 0,C 180,E1 -11613.109,E2 -11613.109} C_VEL
LIN {X 0,Y 388.736,Z 548.692,A -85,B 0,C 180,E1 -11614.666,E2 -11614.666} C_VEL
LIN {X 0,Y 388.795,Z 545.129,A -85,B 0,C 180,E1 -11616.226,E2 -11616.226} C_VEL
LIN {X 0,Y 388.986,Z 540.445,A -85,B 0,C 180,E1 -11617.787,E2 -11617.787} C_VEL
LIN {X 0,Y 389.384,Z 533.368,A -85,B 0,C 180,E1 -11619.61,E2 -11619.61} C_VEL
LIN {X 0,Y 389.89,Z 525.695,A -85,B 0,C 180,E1 -11621.173,E2 -11621.173} C_VEL
LIN {X 0,Y 390.568,Z 517.843,A -85,B 0,C 180,E1 -11622.47,E2 -11622.47} C_VEL
LIN {X 0,Y 391.37,Z 507.791,A -85,B 0,C 180,E1 -11623.819,E2 -11623.819} C_VEL
LIN {X 0,Y 392.037,Z 497.553,A -85,B 0,C 180,E1 -11624.933,E2 -11624.933} C_VEL
LIN {X 0,Y 392.893,Z 485.598,A -85,B 0,C 180,E1 -11625.963,E2 -11625.963} C_VEL
LIN {X 0,Y 393.769,Z 472.773,A -85,B 0,C 180,E1 -11626.792,E2 -11626.792} C_VEL
LIN {X 0,Y 394.38,Z 459.862,A -85,B 0,C 180,E1 -11627.4,E2 -11627.4} C_VEL
LIN {X 0,Y 394.864,Z 447.234,A -85,B 0,C 180,E1 -11627.779,E2 -11627.779} C_VEL
LIN {X 0,Y 395.741,Z 370.22,A -85,B 0,C 180,E1 -11629.185,E2 -11629.185} C_VEL
LIN {X 0,Y 391.539,Z 340.602,A -85,B 0,C 180,E1 -11629.94,E2 -11629.94} C_VEL
LIN {X 0,Y 392.763,Z 323.364,A -85,B 0,C 180,E1 -11633.461,E2 -11633.461} C_VEL
LIN {X 0,Y 393.005,Z 316.68,A -85,B 0,C 180,E1 -11634.849,E2 -11634.849} C_VEL
LIN {X 0,Y 390.674,Z 304.375,A -85,B 0,C 180,E1 -11637.595,E2 -11637.595} C_VEL
LIN {X 0,Y 390.183,Z 301.886,A -85,B 0,C 180,E1 -11638.185,E2 -11638.185} C_VEL
LIN {X 0,Y 390.032,Z 301.904,A -85,B 0,C 180,E1 -11642.124,E2 -11642.124} C_VEL
LIN {X 0,Y 390.084,Z 301.89,A -85,B 0,C 180,E1 -11645.206,E2 -11645.206} C_VEL
LIN {X 0,Y 390.066,Z 301.892,A -85,B 0,C 180,E1 -11649.217,E2 -11649.217} C_VEL
LIN {X 0,Y 390.041,Z 301.902,A -85,B 0,C 180,E1 -11652.373,E2 -11652.373} C_VEL
LIN {X 0,Y 390.042,Z 301.895,A -85,B 0,C 180,E1 -11655.354,E2 -11655.354} C_VEL
LIN {X 0,Y 390.029,Z 301.9,A -85,B 0,C 180,E1 -11658.186,E2 -11658.186} C_VEL
LIN {X 0,Y 390.088,Z 301.894,A -85,B 0,C 180,E1 -11660.907,E2 -11660.907} C_VEL
LIN {X 0,Y 390.082,Z 301.898,A -85,B 0,C 180,E1 -11664.792,E2 -11664.792} C_VEL
LIN {X 0,Y 390.02,Z 301.901,A -85,B 0,C 180,E1 -11668.495,E2 -11668.495} C_VEL
LIN {X 0,Y 390.114,Z 301.886,A -85,B 0,C 180,E1 -11672.069,E2 -11672.069} C_VEL
LIN {X 0,Y 390.076,Z 301.893,A -85,B 0,C 180,E1 -11675.519,E2 -11675.519} C_VEL
LIN {X 0,Y 390.051,Z 301.898,A -85,B 0,C 180,E1 -11678.877,E2 -11678.877} C_VEL
LIN {X 0,Y 390.124,Z 301.885,A -85,B 0,C 180,E1 -11682.166,E2 -11682.166} C_VEL
LIN {X 0,Y 390.14,Z 301.89,A -85,B 0,C 180,E1 -11685.392,E2 -11685.392} C_VEL
LIN {X 0,Y 390.143,Z 301.883,A -85,B 0,C 180,E1 -11688.571,E2 -11688.571} C_VEL
LIN {X 0,Y 390.303,Z 301.864,A -85,B 0,C 180,E1 -11692.031,E2 -11692.031} C_VEL
LIN {X 0,Y 390.22,Z 301.873,A -85,B 0,C 180,E1 -11694.833,E2 -11694.833} C_VEL
LIN {X 0,Y 390.412,Z 301.853,A -85,B 0,C 180,E1 -11697.937,E2 -11697.937} C_VEL
LIN {X 0,Y 390.542,Z 301.837,A -85,B 0,C 180,E1 -11700,E2 -11700} C_VEL
LIN {X 0,Y 390.306,Z 301.863,A -85,B 0,C 180,E1 -11703.096,E2 -11703.096} C_VEL
LIN {X 0,Y 390.278,Z 301.867,A -85,B 0,C 180,E1 -11706.496,E2 -11706.496} C_VEL
LIN {X 0,Y 390.199,Z 301.877,A -85,B 0,C 180,E1 -11709.329,E2 -11709.329} C_VEL
LIN {X 0,Y 390.189,Z 301.878,A -85,B 0,C 180,E1 -11713.438,E2 -11713.438} C_VEL
LIN {X 0,Y 390.143,Z 301.883,A -85,B 0,C 180,E1 -11717.308,E2 -11717.308} C_VEL
LIN {X 0,Y 390.082,Z 301.895,A -85,B 0,C 180,E1 -11720.47,E2 -11720.47} C_VEL
LIN {X 0,Y 390.07,Z 301.898,A -85,B 0,C 180,E1 -11724.481,E2 -11724.481} C_VEL
LIN {X 0,Y 390.112,Z 301.888,A -85,B 0,C 180,E1 -11727.93,E2 -11727.93} C_VEL
LIN {X 0,Y 390.018,Z 301.898,A -85,B 0,C 180,E1 -11731.505,E2 -11731.505} C_VEL
LIN {X 0,Y 390.08,Z 301.892,A -85,B 0,C 180,E1 -11735.207,E2 -11735.207} C_VEL
LIN {X 0,Y 390.062,Z 301.895,A -85,B 0,C 180,E1 -11739.218,E2 -11739.218} C_VEL
LIN {X 0,Y 390.037,Z 301.898,A -85,B 0,C 180,E1 -11742.374,E2 -11742.374} C_VEL
LIN {X 0,Y 390.039,Z 301.898,A -85,B 0,C 180,E1 -11745.355,E2 -11745.355} C_VEL
LIN {X 0,Y 390.013,Z 301.899,A -85,B 0,C 180,E1 -11748.185,E2 -11748.185} C_VEL
LIN {X 0,Y 390.055,Z 301.898,A -85,B 0,C 180,E1 -11750.904,E2 -11750.904} C_VEL
LIN {X 0,Y 390.081,Z 301.893,A -85,B 0,C 180,E1 -11754.794,E2 -11754.794} C_VEL
LIN {X 0,Y 390.02,Z 301.898,A -85,B 0,C 180,E1 -11758.496,E2 -11758.496} C_VEL
LIN {X 0,Y 390.012,Z 301.9,A -85,B 0,C 180,E1 -11762.003,E2 -11762.003} C_VEL
LIN {X 0,Y 390.041,Z 301.903,A -85,B 0,C 180,E1 -11765.517,E2 -11765.517} C_VEL
LIN {X 0,Y 390.059,Z 301.894,A -85,B 0,C 180,E1 -11768.879,E2 -11768.879} C_VEL
LIN {X 0,Y 390.109,Z 301.889,A -85,B 0,C 180,E1 -11772.166,E2 -11772.166} C_VEL
LIN {X 0,Y 390.142,Z 301.886,A -85,B 0,C 180,E1 -11775.393,E2 -11775.393} C_VEL
LIN {X 0,Y 390.241,Z 301.993,A -85,B 0,C 180,E1 -11777.408,E2 -11777.408} C_VEL
LIN {X 0,Y 391.973,Z 312.485,A -85,B 0,C 180,E1 -11779.937,E2 -11779.937} C_VEL
LIN {X 0,Y 392.006,Z 313.484,A -85,B 0,C 180,E1 -11780.168,E2 -11780.168} C_VEL
LIN {X 0,Y 396.158,Z 336.636,A -85,B 0,C 180,E1 -11780.793,E2 -11780.793} C_VEL
LIN {X 0,Y 394.98,Z 420.789,A -85,B 0,C 180,E1 -11782.331,E2 -11782.331} C_VEL
LIN {X 0,Y 394.573,Z 433.965,A -85,B 0,C 180,E1 -11782.774,E2 -11782.774} C_VEL
LIN {X 0,Y 394.079,Z 446.59,A -85,B 0,C 180,E1 -11783.408,E2 -11783.408} C_VEL
LIN {X 0,Y 393.442,Z 458.643,A -85,B 0,C 180,E1 -11784.234,E2 -11784.234} C_VEL
LIN {X 0,Y 392.677,Z 467.563,A -85,B 0,C 180,E1 -11784.995,E2 -11784.995} C_VEL
LIN {X 0,Y 391.894,Z 478.326,A -85,B 0,C 180,E1 -11786.144,E2 -11786.144} C_VEL
LIN {X 0,Y 391.108,Z 488.011,A -85,B 0,C 180,E1 -11787.426,E2 -11787.426} C_VEL
LIN {X 0,Y 390.533,Z 495.942,A -85,B 0,C 180,E1 -11788.711,E2 -11788.711} C_VEL
LIN {X 0,Y 389.87,Z 503.747,A -85,B 0,C 180,E1 -11790.259,E2 -11790.259} C_VEL
LIN {X 0,Y 389.469,Z 509.04,A -85,B 0,C 180,E1 -11791.551,E2 -11791.551} C_VEL
LIN {X 0,Y 389.199,Z 514.21,A -85,B 0,C 180,E1 -11793.106,E2 -11793.106} C_VEL
LIN {X 0,Y 388.936,Z 518.24,A -85,B 0,C 180,E1 -11794.664,E2 -11794.664} C_VEL
LIN {X 0,Y 388.919,Z 521.409,A -85,B 0,C 180,E1 -11796.342,E2 -11796.342} C_VEL
LIN {X 0,Y 388.823,Z 522.096,A -85,B 0,C 180,E1 -11796.845,E2 -11796.845} C_VEL
LIN {X 0,Y 388.038,Z 523.176,A -85,B 0,C 180,E1 -11797.694,E2 -11797.694} C_VEL
LIN {X 0,Y 385.048,Z 524.342,A -85,B 0,C 180,E1 -11799.085,E2 -11799.085} C_VEL
LIN {X 0,Y 382.609,Z 524.786,A -85,B 0,C 180,E1 -11800.216,E2 -11800.216} C_VEL
LIN {X 0,Y 381.614,Z 524.795,A -85,B 0,C 180,E1 -11801.093,E2 -11801.093} C_VEL
LIN {X 0,Y 381.558,Z 524.69,A -85,B 0,C 180,E1 -11801.39,E2 -11801.39} C_VEL
LIN {X 0,Y 381.673,Z 523.99,A -85,B 0,C 180,E1 -11802.766,E2 -11802.766} C_VEL
LIN {X 0,Y 381.732,Z 522.962,A -85,B 0,C 180,E1 -11803.848,E2 -11803.848} C_VEL
LIN {X 0,Y 381.876,Z 521.478,A -85,B 0,C 180,E1 -11804.931,E2 -11804.931} C_VEL
LIN {X 0,Y 382.224,Z 518.42,A -85,B 0,C 180,E1 -11806.559,E2 -11806.559} C_VEL
LIN {X 0,Y 382.637,Z 514.254,A -85,B 0,C 180,E1 -11808.195,E2 -11808.195} C_VEL
LIN {X 0,Y 383.389,Z 507.82,A -85,B 0,C 180,E1 -11810.103,E2 -11810.103} C_VEL
LIN {X 0,Y 384.158,Z 500.744,A -85,B 0,C 180,E1 -11811.744,E2 -11811.744} C_VEL
LIN {X 0,Y 385.204,Z 491.783,A -85,B 0,C 180,E1 -11813.38,E2 -11813.38} C_VEL
LIN {X 0,Y 386.232,Z 482.533,A -85,B 0,C 180,E1 -11814.741,E2 -11814.741} C_VEL
LIN {X 0,Y 387.305,Z 472.228,A -85,B 0,C 180,E1 -11815.962,E2 -11815.962} C_VEL
LIN {X 0,Y 388.358,Z 461.108,A -85,B 0,C 180,E1 -11817.005,E2 -11817.005} C_VEL
LIN {X 0,Y 389.207,Z 449.437,A -85,B 0,C 180,E1 -11817.866,E2 -11817.866} C_VEL
LIN {X 0,Y 389.903,Z 437.403,A -85,B 0,C 180,E1 -11818.533,E2 -11818.533} C_VEL
LIN {X 0,Y 390.238,Z 424.858,A -85,B 0,C 180,E1 -11819.021,E2 -11819.021} C_VEL
LIN {X 0,Y 390.751,Z 409.093,A -85,B 0,C 180,E1 -11819.362,E2 -11819.362} C_VEL
LIN {X 0,Y 392.009,Z 337.414,A -85,B 0,C 180,E1 -11820.691,E2 -11820.691} C_VEL
LIN {X 0,Y 388.089,Z 320.786,A -85,B 0,C 180,E1 -11821.281,E2 -11821.281} C_VEL
LIN {X 0,Y 385.496,Z 313.969,A -85,B 0,C 180,E1 -11821.604,E2 -11821.604} C_VEL
LIN {X 0,Y 383.07,Z 302.772,A -85,B 0,C 180,E1 -11824.559,E2 -11824.559} C_VEL
LIN {X 0,Y 382.998,Z 302.769,A -85,B 0,C 180,E1 -11827.904,E2 -11827.904} C_VEL
LIN {X 0,Y 382.983,Z 302.778,A -85,B 0,C 180,E1 -11831.348,E2 -11831.348} C_VEL
LIN {X 0,Y 382.995,Z 302.776,A -85,B 0,C 180,E1 -11834.303,E2 -11834.303} C_VEL
LIN {X 0,Y 383.009,Z 302.774,A -85,B 0,C 180,E1 -11837.24,E2 -11837.24} C_VEL
LIN {X 0,Y 383.015,Z 302.774,A -85,B 0,C 180,E1 -11840.414,E2 -11840.414} C_VEL
LIN {X 0,Y 383.024,Z 302.768,A -85,B 0,C 180,E1 -11844.045,E2 -11844.045} C_VEL
LIN {X 0,Y 382.986,Z 302.772,A -85,B 0,C 180,E1 -11847.578,E2 -11847.578} C_VEL
LIN {X 0,Y 382.991,Z 302.769,A -85,B 0,C 180,E1 -11850.3,E2 -11850.3} C_VEL
LIN {X 0,Y 383.079,Z 302.76,A -85,B 0,C 180,E1 -11854.021,E2 -11854.021} C_VEL
LIN {X 0,Y 382.994,Z 302.772,A -85,B 0,C 180,E1 -11857.335,E2 -11857.335} C_VEL
LIN {X 0,Y 383.06,Z 302.759,A -85,B 0,C 180,E1 -11860.717,E2 -11860.717} C_VEL
LIN {X 0,Y 383.08,Z 302.76,A -85,B 0,C 180,E1 -11864.027,E2 -11864.027} C_VEL
LIN {X 0,Y 383.136,Z 302.76,A -85,B 0,C 180,E1 -11867.284,E2 -11867.284} C_VEL
LIN {X 0,Y 383.151,Z 302.755,A -85,B 0,C 180,E1 -11870.498,E2 -11870.498} C_VEL
LIN {X 0,Y 383.271,Z 302.737,A -85,B 0,C 180,E1 -11872.625,E2 -11872.625} C_VEL
LIN {X 0,Y 383.197,Z 302.747,A -85,B 0,C 180,E1 -11874.739,E2 -11874.739} C_VEL
LIN {X 0,Y 383.385,Z 302.723,A -85,B 0,C 180,E1 -11877.899,E2 -11877.899} C_VEL
LIN {X 0,Y 383.517,Z 302.713,A -85,B 0,C 180,E1 -11880,E2 -11880} C_VEL
LIN {X 0,Y 383.246,Z 302.737,A -85,B 0,C 180,E1 -11883.154,E2 -11883.154} C_VEL
LIN {X 0,Y 383.285,Z 302.735,A -85,B 0,C 180,E1 -11886.317,E2 -11886.317} C_VEL
LIN {X 0,Y 383.26,Z 302.742,A -85,B 0,C 180,E1 -11888.436,E2 -11888.436} C_VEL
LIN {X 0,Y 383.097,Z 302.755,A -85,B 0,C 180,E1 -11891.642,E2 -11891.642} C_VEL
LIN {X 0,Y 383.11,Z 302.758,A -85,B 0,C 180,E1 -11894.882,E2 -11894.882} C_VEL
LIN {X 0,Y 383.09,Z 302.763,A -85,B 0,C 180,E1 -11898.173,E2 -11898.173} C_VEL
LIN {X 0,Y 382.993,Z 302.773,A -85,B 0,C 180,E1 -11901.531,E2 -11901.531} C_VEL
LIN {X 0,Y 383.052,Z 302.767,A -85,B 0,C 180,E1 -11904.961,E2 -11904.961} C_VEL
LIN {X 0,Y 383.041,Z 302.768,A -85,B 0,C 180,E1 -11908.493,E2 -11908.493} C_VEL
LIN {X 0,Y 383.01,Z 302.769,A -85,B 0,C 180,E1 -11912.15,E2 -11912.15} C_VEL
LIN {X 0,Y 383.019,Z 302.774,A -85,B 0,C 180,E1 -11914.668,E2 -11914.668} C_VEL
LIN {X 0,Y 383,Z 302.773,A -85,B 0,C 180,E1 -11917.904,E2 -11917.904} C_VEL
LIN {X 0,Y 382.985,Z 302.765,A -85,B 0,C 180,E1 -11921.348,E2 -11921.348} C_VEL
LIN {X 0,Y 382.997,Z 302.772,A -85,B 0,C 180,E1 -11924.303,E2 -11924.303} C_VEL
LIN {X 0,Y 383.012,Z 302.775,A -85,B 0,C 180,E1 -11927.24,E2 -11927.24} C_VEL
LIN {X 0,Y 383.015,Z 302.772,A -85,B 0,C 180,E1 -11930.414,E2 -11930.414} C_VEL
LIN {X 0,Y 383.027,Z 302.776,A -85,B 0,C 180,E1 -11934.045,E2 -11934.045} C_VEL
LIN {X 0,Y 382.989,Z 302.777,A -85,B 0,C 180,E1 -11937.578,E2 -11937.578} C_VEL
LIN {X 0,Y 383.005,Z 302.779,A -85,B 0,C 180,E1 -11939.888,E2 -11939.888} C_VEL
LIN {X 0,Y 385.545,Z 313.561,A -85,B 0,C 180,E1 -11942.595,E2 -11942.595} C_VEL
LIN {X 0,Y 387.268,Z 322.596,A -85,B 0,C 180,E1 -11944.757,E2 -11944.757} C_VEL
LIN {X 0,Y 386.07,Z 336.595,A -85,B 0,C 180,E1 -11947.758,E2 -11947.758} C_VEL
LIN {X 0,Y 385.813,Z 340,A -85,B 0,C 180,E1 -11948.483,E2 -11948.483} C_VEL
LIN {X 0,Y 390.504,Z 365.042,A -85,B 0,C 180,E1 -11949.289,E2 -11949.289} C_VEL
LIN {X 0,Y 391.585,Z 372.975,A -85,B 0,C 180,E1 -11949.513,E2 -11949.513} C_VEL
LIN {X 0,Y 390.288,Z 449.198,A -85,B 0,C 180,E1 -11950.958,E2 -11950.958} C_VEL
LIN {X 0,Y 389.512,Z 462.794,A -85,B 0,C 180,E1 -11951.423,E2 -11951.423} C_VEL
LIN {X 0,Y 388.666,Z 475.713,A -85,B 0,C 180,E1 -11952.097,E2 -11952.097} C_VEL
LIN {X 0,Y 387.512,Z 488.254,A -85,B 0,C 180,E1 -11952.995,E2 -11952.995} C_VEL
LIN {X 0,Y 386.382,Z 499.444,A -85,B 0,C 180,E1 -11954.031,E2 -11954.031} C_VEL
LIN {X 0,Y 385.308,Z 509.545,A -85,B 0,C 180,E1 -11955.205,E2 -11955.205} C_VEL
LIN {X 0,Y 384.43,Z 518.667,A -85,B 0,C 180,E1 -11956.521,E2 -11956.521} C_VEL
LIN {X 0,Y 383.381,Z 527.577,A -85,B 0,C 180,E1 -11958.098,E2 -11958.098} C_VEL
LIN {X 0,Y 382.664,Z 534.769,A -85,B 0,C 180,E1 -11959.684,E2 -11959.684} C_VEL
LIN {X 0,Y 382.092,Z 541.343,A -85,B 0,C 180,E1 -11961.538,E2 -11961.538} C_VEL
LIN {X 0,Y 381.781,Z 545.71,A -85,B 0,C 180,E1 -11963.128,E2 -11963.128} C_VEL
LIN {X 0,Y 381.644,Z 549.019,A -85,B 0,C 180,E1 -11964.717,E2 -11964.717} C_VEL
LIN {X 0,Y 381.626,Z 550.673,A -85,B 0,C 180,E1 -11965.775,E2 -11965.775} C_VEL
LIN {X 0,Y 381.549,Z 551.925,A -85,B 0,C 180,E1 -11966.832,E2 -11966.832} C_VEL
LIN {X 0,Y 381.599,Z 552.77,A -85,B 0,C 180,E1 -11967.889,E2 -11967.889} C_VEL
LIN {X 0,Y 381.64,Z 553.187,A -85,B 0,C 180,E1 -11968.944,E2 -11968.944} C_VEL
LIN {X 0,Y 381.656,Z 553.216,A -85,B 0,C 180,E1 -11970,E2 -11970} C_VEL
LIN {X 0,Y 381.672,Z 552.859,A -85,B 0,C 180,E1 -11971.055,E2 -11971.055} C_VEL
LIN {X 0,Y 381.624,Z 552.1,A -85,B 0,C 180,E1 -11972.11,E2 -11972.11} C_VEL
LIN {X 0,Y 381.636,Z 549.284,A -85,B 0,C 180,E1 -11974.224,E2 -11974.224} C_VEL
LIN {X 0,Y 381.688,Z 545.305,A -85,B 0,C 180,E1 -11976.118,E2 -11976.118} C_VEL
LIN {X 0,Y 381.908,Z 540.005,A -85,B 0,C 180,E1 -11977.933,E2 -11977.933} C_VEL
LIN {X 0,Y 382.328,Z 532.884,A -85,B 0,C 180,E1 -11979.789,E2 -11979.789} C_VEL
LIN {X 0,Y 382.893,Z 525.152,A -85,B 0,C 180,E1 -11981.38,E2 -11981.38} C_VEL
LIN {X 0,Y 383.566,Z 517.225,A -85,B 0,C 180,E1 -11982.701,E2 -11982.701} C_VEL
LIN {X 0,Y 384.356,Z 508.082,A -85,B 0,C 180,E1 -11983.953,E2 -11983.953} C_VEL
LIN {X 0,Y 385.077,Z 496.758,A -85,B 0,C 180,E1 -11985.209,E2 -11985.209} C_VEL
LIN {X 0,Y 385.902,Z 486.345,A -85,B 0,C 180,E1 -11986.124,E2 -11986.124} C_VEL
LIN {X 0,Y 386.763,Z 473.852,A -85,B 0,C 180,E1 -11986.97,E2 -11986.97} C_VEL
LIN {X 0,Y 387.471,Z 460.665,A -85,B 0,C 180,E1 -11987.618,E2 -11987.618} C_VEL
LIN {X 0,Y 388.011,Z 447.534,A -85,B 0,C 180,E1 -11988.036,E2 -11988.036} C_VEL
LIN {X 0,Y 388.935,Z 371.005,A -85,B 0,C 180,E1 -11989.459,E2 -11989.459} C_VEL
LIN {X 0,Y 384.592,Z 340.436,A -85,B 0,C 180,E1 -11990.237,E2 -11990.237} C_VEL
LIN {X 0,Y 385.889,Z 323.112,A -85,B 0,C 180,E1 -11993.839,E2 -11993.839} C_VEL
LIN {X 0,Y 386.133,Z 318.8,A -85,B 0,C 180,E1 -11994.747,E2 -11994.747} C_VEL
LIN {X 0,Y 384.131,Z 307.874,A -85,B 0,C 180,E1 -11997.219,E2 -11997.219} C_VEL
LIN {X 0,Y 383.109,Z 302.768,A -85,B 0,C 180,E1 -11998.414,E2 -11998.414} C_VEL
LIN {X 0,Y 382.987,Z 302.778,A -85,B 0,C 180,E1 -12002.421,E2 -12002.421} C_VEL
LIN {X 0,Y 383.024,Z 302.773,A -85,B 0,C 180,E1 -12005.955,E2 -12005.955} C_VEL
LIN {X 0,Y 383.012,Z 302.771,A -85,B 0,C 180,E1 -12009.585,E2 -12009.585} C_VEL
LIN {X 0,Y 383.004,Z 302.775,A -85,B 0,C 180,E1 -12012.778,E2 -12012.778} C_VEL
LIN {X 0,Y 382.995,Z 302.774,A -85,B 0,C 180,E1 -12015.788,E2 -12015.788} C_VEL
LIN {X 0,Y 382.986,Z 302.779,A -85,B 0,C 180,E1 -12018.795,E2 -12018.795} C_VEL
LIN {X 0,Y 382.997,Z 302.774,A -85,B 0,C 180,E1 -12022.096,E2 -12022.096} C_VEL
LIN {X 0,Y 383.015,Z 302.772,A -85,B 0,C 180,E1 -12025.331,E2 -12025.331} C_VEL
LIN {X 0,Y 382.979,Z 302.78,A -85,B 0,C 180,E1 -12029.081,E2 -12029.081} C_VEL
LIN {X 0,Y 383.053,Z 302.77,A -85,B 0,C 180,E1 -12032.698,E2 -12032.698} C_VEL
LIN {X 0,Y 383.048,Z 302.774,A -85,B 0,C 180,E1 -12035.039,E2 -12035.039} C_VEL
LIN {X 0,Y 382.989,Z 302.775,A -85,B 0,C 180,E1 -12038.469,E2 -12038.469} C_VEL
LIN {X 0,Y 383.085,Z 302.763,A -85,B 0,C 180,E1 -12041.827,E2 -12041.827} C_VEL
LIN {X 0,Y 383.106,Z 302.764,A -85,B 0,C 180,E1 -12045.118,E2 -12045.118} C_VEL
LIN {X 0,Y 383.093,Z 302.761,A -85,B 0,C 180,E1 -12048.358,E2 -12048.358} C_VEL
LIN {X 0,Y 383.259,Z 302.742,A -85,B 0,C 180,E1 -12051.975,E2 -12051.975} C_VEL
LIN {X 0,Y 383.192,Z 302.749,A -85,B 0,C 180,E1 -12054.738,E2 -12054.738} C_VEL
LIN {X 0,Y 383.38,Z 302.73,A -85,B 0,C 180,E1 -12057.899,E2 -12057.899} C_VEL
LIN {X 0,Y 383.512,Z 302.713,A -85,B 0,C 180,E1 -12060,E2 -12060} C_VEL
LIN {X 0,Y 383.242,Z 302.743,A -85,B 0,C 180,E1 -12063.153,E2 -12063.153} C_VEL
LIN {X 0,Y 383.241,Z 302.744,A -85,B 0,C 180,E1 -12066.482,E2 -12066.482} C_VEL
LIN {X 0,Y 383.145,Z 302.756,A -85,B 0,C 180,E1 -12069.502,E2 -12069.502} C_VEL
LIN {X 0,Y 383.12,Z 302.759,A -85,B 0,C 180,E1 -12073.536,E2 -12073.536} C_VEL
LIN {X 0,Y 383.089,Z 302.762,A -85,B 0,C 180,E1 -12077.454,E2 -12077.454} C_VEL
LIN {X 0,Y 383.023,Z 302.773,A -85,B 0,C 180,E1 -12080.647,E2 -12080.647} C_VEL
LIN {X 0,Y 383.016,Z 302.772,A -85,B 0,C 180,E1 -12083.808,E2 -12083.808} C_VEL
LIN {X 0,Y 383.074,Z 302.767,A -85,B 0,C 180,E1 -12086.124,E2 -12086.124} C_VEL
LIN {X 0,Y 383.035,Z 302.776,A -85,B 0,C 180,E1 -12088.493,E2 -12088.493} C_VEL
LIN {X 0,Y 383.004,Z 302.774,A -85,B 0,C 180,E1 -12092.15,E2 -12092.15} C_VEL
LIN {X 0,Y 383.013,Z 302.778,A -85,B 0,C 180,E1 -12094.668,E2 -12094.668} C_VEL
LIN {X 0,Y 382.993,Z 302.773,A -85,B 0,C 180,E1 -12097.904,E2 -12097.904} C_VEL
LIN {X 0,Y 382.979,Z 302.777,A -85,B 0,C 180,E1 -12101.348,E2 -12101.348} C_VEL
LIN {X 0,Y 382.991,Z 302.775,A -85,B 0,C 180,E1 -12104.304,E2 -12104.304} C_VEL
LIN {X 0,Y 383.006,Z 302.776,A -85,B 0,C 180,E1 -12107.241,E2 -12107.241} C_VEL
LIN {X 0,Y 382.982,Z 302.775,A -85,B 0,C 180,E1 -12110.419,E2 -12110.419} C_VEL
LIN {X 0,Y 383.021,Z 302.77,A -85,B 0,C 180,E1 -12114.045,E2 -12114.045} C_VEL
LIN {X 0,Y 382.983,Z 302.778,A -85,B 0,C 180,E1 -12117.579,E2 -12117.579} C_VEL
LIN {X 0,Y 382.973,Z 302.776,A -85,B 0,C 180,E1 -12120.299,E2 -12120.299} C_VEL
LIN {X 0,Y 383,Z 302.774,A -85,B 0,C 180,E1 -12124.045,E2 -12124.045} C_VEL
LIN {X 0,Y 382.986,Z 302.779,A -85,B 0,C 180,E1 -12127.334,E2 -12127.334} C_VEL
LIN {X 0,Y 383.057,Z 302.765,A -85,B 0,C 180,E1 -12130.717,E2 -12130.717} C_VEL
LIN {X 0,Y 383.079,Z 302.768,A -85,B 0,C 180,E1 -12134.027,E2 -12134.027} C_VEL
LIN {X 0,Y 383.204,Z 302.87,A -85,B 0,C 180,E1 -12137.184,E2 -12137.184} C_VEL
LIN {X 0,Y 385.019,Z 313.749,A -85,B 0,C 180,E1 -12139.856,E2 -12139.856} C_VEL
LIN {X 0,Y 389.357,Z 337.445,A -85,B 0,C 180,E1 -12140.509,E2 -12140.509} C_VEL
LIN {X 0,Y 388.143,Z 421.078,A -85,B 0,C 180,E1 -12142.065,E2 -12142.065} C_VEL
LIN {X 0,Y 387.721,Z 434.243,A -85,B 0,C 180,E1 -12142.514,E2 -12142.514} C_VEL
LIN {X 0,Y 387.207,Z 446.865,A -85,B 0,C 180,E1 -12143.16,E2 -12143.16} C_VEL
LIN {X 0,Y 386.547,Z 458.913,A -85,B 0,C 180,E1 -12144,E2 -12144} C_VEL
LIN {X 0,Y 385.765,Z 467.831,A -85,B 0,C 180,E1 -12144.774,E2 -12144.774} C_VEL
LIN {X 0,Y 384.944,Z 478.595,A -85,B 0,C 180,E1 -12145.944,E2 -12145.944} C_VEL
LIN {X 0,Y 384.182,Z 487.397,A -85,B 0,C 180,E1 -12147.117,E2 -12147.117} C_VEL
LIN {X 0,Y 383.469,Z 496.948,A -85,B 0,C 180,E1 -12148.688,E2 -12148.688} C_VEL
LIN {X 0,Y 382.781,Z 504.574,A -85,B 0,C 180,E1 -12150.263,E2 -12150.263} C_VEL
LIN {X 0,Y 382.32,Z 511.594,A -85,B 0,C 180,E1 -12152.107,E2 -12152.107} C_VEL
LIN {X 0,Y 381.966,Z 516.279,A -85,B 0,C 180,E1 -12153.693,E2 -12153.693} C_VEL
LIN {X 0,Y 381.865,Z 519.854,A -85,B 0,C 180,E1 -12155.28,E2 -12155.28} C_VEL
LIN {X 0,Y 381.742,Z 522.306,A -85,B 0,C 180,E1 -12156.808,E2 -12156.808} C_VEL
LIN {X 0,Y 381.563,Z 524.076,A -85,B 0,C 180,E1 -12158.474,E2 -12158.474} C_VEL
LIN {X 0,Y 381.502,Z 524.677,A -85,B 0,C 180,E1 -12159.544,E2 -12159.544} C_VEL
LIN {X 0,Y 381.558,Z 524.69,A -85,B 0,C 180,E1 -12161.39,E2 -12161.39} C_VEL
LIN {X 0,Y 380.963,Z 524.386,A -85,B 0,C 180,E1 -12162.27,E2 -12162.27} C_VEL
LIN {X 0,Y 378.195,Z 523.313,A -85,B 0,C 180,E1 -12163.698,E2 -12163.698} C_VEL
LIN {X 0,Y 375.491,Z 521.621,A -85,B 0,C 180,E1 -12165.131,E2 -12165.131} C_VEL
LIN {X 0,Y 375.016,Z 520.103,A -85,B 0,C 180,E1 -12166.006,E2 -12166.006} C_VEL
LIN {X 0,Y 375.377,Z 517.102,A -85,B 0,C 180,E1 -12167.431,E2 -12167.431} C_VEL
LIN {X 0,Y 375.901,Z 512.437,A -85,B 0,C 180,E1 -12169.098,E2 -12169.098} C_VEL
LIN {X 0,Y 376.633,Z 506.454,A -85,B 0,C 180,E1 -12170.766,E2 -12170.766} C_VEL
LIN {X 0,Y 377.487,Z 498.928,A -85,B 0,C 180,E1 -12172.437,E2 -12172.437} C_VEL
LIN {X 0,Y 378.487,Z 491.211,A -85,B 0,C 180,E1 -12173.82,E2 -12173.82} C_VEL
LIN {X 0,Y 379.613,Z 481.785,A -85,B 0,C 180,E1 -12175.202,E2 -12175.202} C_VEL
LIN {X 0,Y 380.724,Z 471.174,A -85,B 0,C 180,E1 -12176.445,E2 -12176.445} C_VEL
LIN {X 0,Y 381.719,Z 460.944,A -85,B 0,C 180,E1 -12177.406,E2 -12177.406} C_VEL
LIN {X 0,Y 382.618,Z 449.384,A -85,B 0,C 180,E1 -12178.265,E2 -12178.265} C_VEL
LIN {X 0,Y 383.351,Z 436.959,A -85,B 0,C 180,E1 -12178.954,E2 -12178.954} C_VEL
LIN {X 0,Y 383.728,Z 424.043,A -85,B 0,C 180,E1 -12179.449,E2 -12179.449} C_VEL
LIN {X 0,Y 384.312,Z 404.446,A -85,B 0,C 180,E1 -12179.856,E2 -12179.856} C_VEL
LIN {X 0,Y 385.494,Z 338.667,A -85,B 0,C 180,E1 -12181.097,E2 -12181.097} C_VEL
LIN {X 0,Y 382.045,Z 323.627,A -85,B 0,C 180,E1 -12181.639,E2 -12181.639} C_VEL
LIN {X 0,Y 378.362,Z 314.26,A -85,B 0,C 180,E1 -12182.101,E2 -12182.101} C_VEL
LIN {X 0,Y 375.984,Z 303.653,A -85,B 0,C 180,E1 -12184.999,E2 -12184.999} C_VEL
LIN {X 0,Y 375.973,Z 303.647,A -85,B 0,C 180,E1 -12188.27,E2 -12188.27} C_VEL
LIN {X 0,Y 375.933,Z 303.656,A -85,B 0,C 180,E1 -12191.601,E2 -12191.601} C_VEL
LIN {X 0,Y 375.926,Z 303.658,A -85,B 0,C 180,E1 -12195.269,E2 -12195.269} C_VEL
LIN {X 0,Y 375.934,Z 303.657,A -85,B 0,C 180,E1 -12198.399,E2 -12198.399} C_VEL
LIN {X 0,Y 375.973,Z 303.646,A -85,B 0,C 180,E1 -12201.73,E2 -12201.73} C_VEL
LIN {X 0,Y 375.979,Z 303.647,A -85,B 0,C 180,E1 -12205.333,E2 -12205.333} C_VEL
LIN {X 0,Y 375.957,Z 303.647,A -85,B 0,C 180,E1 -12208.438,E2 -12208.438} C_VEL
LIN {X 0,Y 375.982,Z 303.64,A -85,B 0,C 180,E1 -12212.14,E2 -12212.14} C_VEL
LIN {X 0,Y 376.005,Z 303.642,A -85,B 0,C 180,E1 -12214.539,E2 -12214.539} C_VEL
LIN {X 0,Y 375.957,Z 303.65,A -85,B 0,C 180,E1 -12218.046,E2 -12218.046} C_VEL
LIN {X 0,Y 376.023,Z 303.642,A -85,B 0,C 180,E1 -12221.474,E2 -12221.474} C_VEL
LIN {X 0,Y 376.058,Z 303.633,A -85,B 0,C 180,E1 -12224.833,E2 -12224.833} C_VEL
LIN {X 0,Y 376.049,Z 303.637,A -85,B 0,C 180,E1 -12228.137,E2 -12228.137} C_VEL
LIN {X 0,Y 376.257,Z 303.616,A -85,B 0,C 180,E1 -12231.878,E2 -12231.878} C_VEL
LIN {X 0,Y 376.169,Z 303.623,A -85,B 0,C 180,E1 -12234.64,E2 -12234.64} C_VEL
LIN {X 0,Y 376.351,Z 303.599,A -85,B 0,C 180,E1 -12237.86,E2 -12237.86} C_VEL
LIN {X 0,Y 376.487,Z 303.588,A -85,B 0,C 180,E1 -12240,E2 -12240} C_VEL
LIN {X 0,Y 376.184,Z 303.616,A -85,B 0,C 180,E1 -12243.213,E2 -12243.213} C_VEL
LIN {X 0,Y 376.244,Z 303.61,A -85,B 0,C 180,E1 -12246.435,E2 -12246.435} C_VEL
LIN {X 0,Y 376.206,Z 303.622,A -85,B 0,C 180,E1 -12248.595,E2 -12248.595} C_VEL
LIN {X 0,Y 376.049,Z 303.633,A -85,B 0,C 180,E1 -12251.864,E2 -12251.864} C_VEL
LIN {X 0,Y 376.058,Z 303.634,A -85,B 0,C 180,E1 -12255.168,E2 -12255.168} C_VEL
LIN {X 0,Y 376.024,Z 303.647,A -85,B 0,C 180,E1 -12258.526,E2 -12258.526} C_VEL
LIN {X 0,Y 375.959,Z 303.65,A -85,B 0,C 180,E1 -12261.955,E2 -12261.955} C_VEL
LIN {X 0,Y 376.006,Z 303.645,A -85,B 0,C 180,E1 -12265.461,E2 -12265.461} C_VEL
LIN {X 0,Y 375.971,Z 303.649,A -85,B 0,C 180,E1 -12269.079,E2 -12269.079} C_VEL
LIN {X 0,Y 375.95,Z 303.651,A -85,B 0,C 180,E1 -12272.829,E2 -12272.829} C_VEL
LIN {X 0,Y 375.958,Z 303.649,A -85,B 0,C 180,E1 -12275.416,E2 -12275.416} C_VEL
LIN {X 0,Y 375.974,Z 303.648,A -85,B 0,C 180,E1 -12278.27,E2 -12278.27} C_VEL
LIN {X 0,Y 375.935,Z 303.646,A -85,B 0,C 180,E1 -12281.601,E2 -12281.601} C_VEL
LIN {X 0,Y 375.928,Z 303.658,A -85,B 0,C 180,E1 -12285.269,E2 -12285.269} C_VEL
LIN {X 0,Y 375.936,Z 303.655,A -85,B 0,C 180,E1 -12288.399,E2 -12288.399} C_VEL
LIN {X 0,Y 375.974,Z 303.652,A -85,B 0,C 180,E1 -12291.73,E2 -12291.73} C_VEL
LIN {X 0,Y 375.982,Z 303.648,A -85,B 0,C 180,E1 -12295.333,E2 -12295.333} C_VEL
LIN {X 0,Y 375.96,Z 303.656,A -85,B 0,C 180,E1 -12298.438,E2 -12298.438} C_VEL
LIN {X 0,Y 375.97,Z 303.721,A -85,B 0,C 180,E1 -12299.479,E2 -12299.479} C_VEL
LIN {X 0,Y 378.337,Z 313.596,A -85,B 0,C 180,E1 -12302.028,E2 -12302.028} C_VEL
LIN {X 0,Y 380.374,Z 323.912,A -85,B 0,C 180,E1 -12304.559,E2 -12304.559} C_VEL
LIN {X 0,Y 379.768,Z 331.661,A -85,B 0,C 180,E1 -12306.265,E2 -12306.265} C_VEL
LIN {X 0,Y 379.011,Z 339.647,A -85,B 0,C 180,E1 -12307.995,E2 -12307.995} C_VEL
LIN {X 0,Y 383.57,Z 363.538,A -85,B 0,C 180,E1 -12308.807,E2 -12308.807} C_VEL
LIN {X 0,Y 385.041,Z 373.989,A -85,B 0,C 180,E1 -12309.114,E2 -12309.114} C_VEL
LIN {X 0,Y 383.728,Z 448.535,A -85,B 0,C 180,E1 -12310.548,E2 -12310.548} C_VEL
LIN {X 0,Y 382.943,Z 462.291,A -85,B 0,C 180,E1 -12311.023,E2 -12311.023} C_VEL
LIN {X 0,Y 382.037,Z 475.282,A -85,B 0,C 180,E1 -12311.706,E2 -12311.706} C_VEL
LIN {X 0,Y 380.896,Z 487.067,A -85,B 0,C 180,E1 -12312.552,E2 -12312.552} C_VEL
LIN {X 0,Y 379.747,Z 498.416,A -85,B 0,C 180,E1 -12313.606,E2 -12313.606} C_VEL
LIN {X 0,Y 378.604,Z 508.675,A -85,B 0,C 180,E1 -12314.799,E2 -12314.799} C_VEL
LIN {X 0,Y 377.709,Z 517.085,A -85,B 0,C 180,E1 -12316.002,E2 -12316.002} C_VEL
LIN {X 0,Y 376.629,Z 526.228,A -85,B 0,C 180,E1 -12317.608,E2 -12317.608} C_VEL
LIN {X 0,Y 375.759,Z 533.609,A -85,B 0,C 180,E1 -12319.22,E2 -12319.22} C_VEL
LIN {X 0,Y 375.194,Z 539.552,A -85,B 0,C 180,E1 -12320.838,E2 -12320.838} C_VEL
LIN {X 0,Y 374.804,Z 544.259,A -85,B 0,C 180,E1 -12322.457,E2 -12322.457} C_VEL
LIN {X 0,Y 374.59,Z 547.566,A -85,B 0,C 180,E1 -12323.925,E2 -12323.925} C_VEL
LIN {X 0,Y 374.552,Z 550.481,A -85,B 0,C 180,E1 -12325.695,E2 -12325.695} C_VEL
LIN {X 0,Y 374.463,Z 551.717,A -85,B 0,C 180,E1 -12326.772,E2 -12326.772} C_VEL
LIN {X 0,Y 374.497,Z 552.529,A -85,B 0,C 180,E1 -12327.849,E2 -12327.849} C_VEL
LIN {X 0,Y 374.556,Z 552.93,A -85,B 0,C 180,E1 -12328.924,E2 -12328.924} C_VEL
LIN {X 0,Y 374.589,Z 552.944,A -85,B 0,C 180,E1 -12330,E2 -12330} C_VEL
LIN {X 0,Y 374.586,Z 552.571,A -85,B 0,C 180,E1 -12331.075,E2 -12331.075} C_VEL
LIN {X 0,Y 374.524,Z 551.782,A -85,B 0,C 180,E1 -12332.15,E2 -12332.15} C_VEL
LIN {X 0,Y 374.565,Z 548.93,A -85,B 0,C 180,E1 -12334.304,E2 -12334.304} C_VEL
LIN {X 0,Y 374.586,Z 545.298,A -85,B 0,C 180,E1 -12336.07,E2 -12336.07} C_VEL
LIN {X 0,Y 374.766,Z 541.269,A -85,B 0,C 180,E1 -12337.543,E2 -12337.543} C_VEL
LIN {X 0,Y 375.073,Z 535.689,A -85,B 0,C 180,E1 -12339.164,E2 -12339.164} C_VEL
LIN {X 0,Y 375.528,Z 528.71,A -85,B 0,C 180,E1 -12340.786,E2 -12340.786} C_VEL
LIN {X 0,Y 376.33,Z 519.963,A -85,B 0,C 180,E1 -12342.401,E2 -12342.401} C_VEL
LIN {X 0,Y 377.118,Z 510.985,A -85,B 0,C 180,E1 -12343.745,E2 -12343.745} C_VEL
LIN {X 0,Y 377.783,Z 501.661,A -85,B 0,C 180,E1 -12344.892,E2 -12344.892} C_VEL
LIN {X 0,Y 378.556,Z 491.7,A -85,B 0,C 180,E1 -12345.892,E2 -12345.892} C_VEL
LIN {X 0,Y 379.464,Z 480,A -85,B 0,C 180,E1 -12346.821,E2 -12346.821} C_VEL
LIN {X 0,Y 380.202,Z 467.809,A -85,B 0,C 180,E1 -12347.549,E2 -12347.549} C_VEL
LIN {X 0,Y 380.928,Z 454.557,A -85,B 0,C 180,E1 -12348.105,E2 -12348.105} C_VEL
LIN {X 0,Y 381.319,Z 441.71,A -85,B 0,C 180,E1 -12348.431,E2 -12348.431} C_VEL
LIN {X 0,Y 382.019,Z 371.271,A -85,B 0,C 180,E1 -12349.758,E2 -12349.758} C_VEL
LIN {X 0,Y 377.67,Z 340.05,A -85,B 0,C 180,E1 -12350.588,E2 -12350.588} C_VEL
LIN {X 0,Y 378.953,Z 323.577,A -85,B 0,C 180,E1 -12354.079,E2 -12354.079} C_VEL
LIN {X 0,Y 379.134,Z 319.7,A -85,B 0,C 180,E1 -12354.914,E2 -12354.914} C_VEL
LIN {X 0,Y 376.817,Z 307.25,A -85,B 0,C 180,E1 -12357.792,E2 -12357.792} C_VEL
LIN {X 0,Y 376.043,Z 303.647,A -85,B 0,C 180,E1 -12358.686,E2 -12358.686} C_VEL
LIN {X 0,Y 375.949,Z 303.652,A -85,B 0,C 180,E1 -12362.729,E2 -12362.729} C_VEL
LIN {X 0,Y 375.957,Z 303.65,A -85,B 0,C 180,E1 -12365.415,E2 -12365.415} C_VEL
LIN {X 0,Y 375.971,Z 303.655,A -85,B 0,C 180,E1 -12368.269,E2 -12368.269} C_VEL
LIN {X 0,Y 375.932,Z 303.653,A -85,B 0,C 180,E1 -12371.6,E2 -12371.6} C_VEL
LIN {X 0,Y 375.925,Z 303.654,A -85,B 0,C 180,E1 -12375.268,E2 -12375.268} C_VEL
LIN {X 0,Y 375.933,Z 303.658,A -85,B 0,C 180,E1 -12378.398,E2 -12378.398} C_VEL
LIN {X 0,Y 375.971,Z 303.648,A -85,B 0,C 180,E1 -12381.729,E2 -12381.729} C_VEL
LIN {X 0,Y 375.977,Z 303.649,A -85,B 0,C 180,E1 -12385.332,E2 -12385.332} C_VEL
LIN {X 0,Y 375.954,Z 303.653,A -85,B 0,C 180,E1 -12388.437,E2 -12388.437} C_VEL
LIN {X 0,Y 375.979,Z 303.647,A -85,B 0,C 180,E1 -12392.14,E2 -12392.14} C_VEL
LIN {X 0,Y 376.002,Z 303.646,A -85,B 0,C 180,E1 -12394.538,E2 -12394.538} C_VEL
LIN {X 0,Y 375.959,Z 303.65,A -85,B 0,C 180,E1 -12398.045,E2 -12398.045} C_VEL
LIN {X 0,Y 376.02,Z 303.646,A -85,B 0,C 180,E1 -12401.474,E2 -12401.474} C_VEL
LIN {X 0,Y 376.054,Z 303.64,A -85,B 0,C 180,E1 -12404.832,E2 -12404.832} C_VEL
LIN {X 0,Y 376.045,Z 303.639,A -85,B 0,C 180,E1 -12408.136,E2 -12408.136} C_VEL
LIN {X 0,Y 376.214,Z 303.62,A -85,B 0,C 180,E1 -12411.918,E2 -12411.918} C_VEL
LIN {X 0,Y 376.165,Z 303.624,A -85,B 0,C 180,E1 -12414.64,E2 -12414.64} C_VEL
LIN {X 0,Y 376.346,Z 303.606,A -85,B 0,C 180,E1 -12417.859,E2 -12417.859} C_VEL
LIN {X 0,Y 376.482,Z 303.588,A -85,B 0,C 180,E1 -12420,E2 -12420} C_VEL
LIN {X 0,Y 376.18,Z 303.623,A -85,B 0,C 180,E1 -12423.213,E2 -12423.213} C_VEL
LIN {X 0,Y 376.211,Z 303.62,A -85,B 0,C 180,E1 -12426.465,E2 -12426.465} C_VEL
LIN {X 0,Y 376.113,Z 303.634,A -85,B 0,C 180,E1 -12429.681,E2 -12429.681} C_VEL
LIN {X 0,Y 376.084,Z 303.636,A -85,B 0,C 180,E1 -12433.658,E2 -12433.658} C_VEL
LIN {X 0,Y 376.039,Z 303.641,A -85,B 0,C 180,E1 -12437.607,E2 -12437.607} C_VEL
LIN {X 0,Y 375.973,Z 303.649,A -85,B 0,C 180,E1 -12440.832,E2 -12440.832} C_VEL
LIN {X 0,Y 375.982,Z 303.653,A -85,B 0,C 180,E1 -12444.282,E2 -12444.282} C_VEL
LIN {X 0,Y 376.014,Z 303.648,A -85,B 0,C 180,E1 -12446.652,E2 -12446.652} C_VEL
LIN {X 0,Y 375.965,Z 303.65,A -85,B 0,C 180,E1 -12449.079,E2 -12449.079} C_VEL
LIN {X 0,Y 375.944,Z 303.656,A -85,B 0,C 180,E1 -12452.829,E2 -12452.829} C_VEL
LIN {X 0,Y 375.952,Z 303.651,A -85,B 0,C 180,E1 -12455.416,E2 -12455.416} C_VEL
LIN {X 0,Y 375.968,Z 303.65,A -85,B 0,C 180,E1 -12458.27,E2 -12458.27} C_VEL
LIN {X 0,Y 375.929,Z 303.654,A -85,B 0,C 180,E1 -12461.601,E2 -12461.601} C_VEL
LIN {X 0,Y 375.921,Z 303.658,A -85,B 0,C 180,E1 -12465.269,E2 -12465.269} C_VEL
LIN {X 0,Y 375.913,Z 303.656,A -85,B 0,C 180,E1 -12468.403,E2 -12468.403} C_VEL
LIN {X 0,Y 375.951,Z 303.651,A -85,B 0,C 180,E1 -12471.911,E2 -12471.911} C_VEL
LIN {X 0,Y 375.976,Z 303.654,A -85,B 0,C 180,E1 -12475.333,E2 -12475.333} C_VEL
LIN {X 0,Y 375.954,Z 303.65,A -85,B 0,C 180,E1 -12478.438,E2 -12478.438} C_VEL
LIN {X 0,Y 375.915,Z 303.656,A -85,B 0,C 180,E1 -12482.135,E2 -12482.135} C_VEL
LIN {X 0,Y 375.956,Z 303.655,A -85,B 0,C 180,E1 -12485.717,E2 -12485.717} C_VEL
LIN {X 0,Y 375.996,Z 303.647,A -85,B 0,C 180,E1 -12489.198,E2 -12489.198} C_VEL
LIN {X 0,Y 376.031,Z 303.641,A -85,B 0,C 180,E1 -12492.601,E2 -12492.601} C_VEL
LIN {X 0,Y 376.096,Z 303.636,A -85,B 0,C 180,E1 -12496.338,E2 -12496.338} C_VEL
LIN {X 0,Y 376.158,Z 303.725,A -85,B 0,C 180,E1 -12496.948,E2 -12496.948} C_VEL
LIN {X 0,Y 377.953,Z 314.091,A -85,B 0,C 180,E1 -12499.527,E2 -12499.527} C_VEL
LIN {X 0,Y 380.195,Z 324.621,A -85,B 0,C 180,E1 -12499.84,E2 -12499.84} C_VEL
LIN {X 0,Y 382.558,Z 338.277,A -85,B 0,C 180,E1 -12500.216,E2 -12500.216} C_VEL
LIN {X 0,Y 381.306,Z 421.371,A -85,B 0,C 180,E1 -12501.788,E2 -12501.788} C_VEL
LIN {X 0,Y 380.881,Z 434.52,A -85,B 0,C 180,E1 -12502.246,E2 -12502.246} C_VEL
LIN {X 0,Y 380.339,Z 447.14,A -85,B 0,C 180,E1 -12502.902,E2 -12502.902} C_VEL
LIN {X 0,Y 379.658,Z 459.184,A -85,B 0,C 180,E1 -12503.757,E2 -12503.757} C_VEL
LIN {X 0,Y 378.841,Z 468.103,A -85,B 0,C 180,E1 -12504.545,E2 -12504.545} C_VEL
LIN {X 0,Y 378,Z 478.863,A -85,B 0,C 180,E1 -12505.735,E2 -12505.735} C_VEL
LIN {X 0,Y 377.149,Z 488.547,A -85,B 0,C 180,E1 -12507.063,E2 -12507.063} C_VEL
LIN {X 0,Y 376.505,Z 496.481,A -85,B 0,C 180,E1 -12508.396,E2 -12508.396} C_VEL
LIN {X 0,Y 375.786,Z 504.286,A -85,B 0,C 180,E1 -12510,E2 -12510} C_VEL
LIN {X 0,Y 375.304,Z 510.515,A -85,B 0,C 180,E1 -12511.61,E2 -12511.61} C_VEL
LIN {X 0,Y 375.011,Z 515.474,A -85,B 0,C 180,E1 -12513.223,E2 -12513.223} C_VEL
LIN {X 0,Y 374.792,Z 519.322,A -85,B 0,C 180,E1 -12514.841,E2 -12514.841} C_VEL
LIN {X 0,Y 374.721,Z 522.148,A -85,B 0,C 180,E1 -12516.462,E2 -12516.462} C_VEL
LIN {X 0,Y 374.459,Z 524.443,A -85,B 0,C 180,E1 -12518.636,E2 -12518.636} C_VEL
LIN {X 0,Y 374.402,Z 524.999,A -85,B 0,C 180,E1 -12519.727,E2 -12519.727} C_VEL
LIN {X 0,Y 374.472,Z 524.959,A -85,B 0,C 180,E1 -12521.406,E2 -12521.406} C_VEL
LIN {X 0,Y 374.596,Z 524.155,A -85,B 0,C 180,E1 -12523.011,E2 -12523.011} C_VEL
LIN {X 0,Y 374.678,Z 523.069,A -85,B 0,C 180,E1 -12524.114,E2 -12524.114} C_VEL
LIN {X 0,Y 375.016,Z 520.103,A -85,B 0,C 180,E1 -12526.006,E2 -12526.006} C_VEL
LIN {X 0,Y 374.584,Z 518.476,A -85,B 0,C 180,E1 -12526.871,E2 -12526.871} C_VEL
LIN {X 0,Y 372.126,Z 515.383,A -85,B 0,C 180,E1 -12528.268,E2 -12528.268} C_VEL
LIN {X 0,Y 369.742,Z 511.614,A -85,B 0,C 180,E1 -12529.641,E2 -12529.641} C_VEL
LIN {X 0,Y 369.433,Z 508.887,A -85,B 0,C 180,E1 -12530.455,E2 -12530.455} C_VEL
LIN {X 0,Y 370.36,Z 501.278,A -85,B 0,C 180,E1 -12532.304,E2 -12532.304} C_VEL
LIN {X 0,Y 371.558,Z 492.325,A -85,B 0,C 180,E1 -12533.996,E2 -12533.996} C_VEL
LIN {X 0,Y 372.817,Z 482.495,A -85,B 0,C 180,E1 -12535.484,E2 -12535.484} C_VEL
LIN {X 0,Y 373.898,Z 472.793,A -85,B 0,C 180,E1 -12536.665,E2 -12536.665} C_VEL
LIN {X 0,Y 375.078,Z 461.241,A -85,B 0,C 180,E1 -12537.781,E2 -12537.781} C_VEL
LIN {X 0,Y 375.992,Z 450.006,A -85,B 0,C 180,E1 -12538.633,E2 -12538.633} C_VEL
LIN {X 0,Y 376.748,Z 438.043,A -85,B 0,C 180,E1 -12539.319,E2 -12539.319} C_VEL
LIN {X 0,Y 377.137,Z 425.568,A -85,B 0,C 180,E1 -12539.823,E2 -12539.823} C_VEL
LIN {X 0,Y 377.708,Z 409.406,A -85,B 0,C 180,E1 -12540.183,E2 -12540.183} C_VEL
LIN {X 0,Y 379.15,Z 340.393,A -85,B 0,C 180,E1 -12541.498,E2 -12541.498} C_VEL
LIN {X 0,Y 375.818,Z 325.865,A -85,B 0,C 180,E1 -12542.036,E2 -12542.036} C_VEL
LIN {X 0,Y 371.166,Z 314.503,A -85,B 0,C 180,E1 -12542.639,E2 -12542.639} C_VEL
LIN {X 0,Y 368.926,Z 304.531,A -85,B 0,C 180,E1 -12545.392,E2 -12545.392} C_VEL
LIN {X 0,Y 368.902,Z 304.536,A -85,B 0,C 180,E1 -12548.953,E2 -12548.953} C_VEL
LIN {X 0,Y 368.88,Z 304.534,A -85,B 0,C 180,E1 -12552.009,E2 -12552.009} C_VEL
LIN {X 0,Y 368.879,Z 304.536,A -85,B 0,C 180,E1 -12555.176,E2 -12555.176} C_VEL
LIN {X 0,Y 368.882,Z 304.534,A -85,B 0,C 180,E1 -12558.178,E2 -12558.178} C_VEL
LIN {X 0,Y 368.908,Z 304.528,A -85,B 0,C 180,E1 -12561.36,E2 -12561.36} C_VEL
LIN {X 0,Y 368.936,Z 304.526,A -85,B 0,C 180,E1 -12565.147,E2 -12565.147} C_VEL
LIN {X 0,Y 368.929,Z 304.521,A -85,B 0,C 180,E1 -12569.047,E2 -12569.047} C_VEL
LIN {X 0,Y 368.975,Z 304.516,A -85,B 0,C 180,E1 -12571.564,E2 -12571.564} C_VEL
LIN {X 0,Y 368.999,Z 304.514,A -85,B 0,C 180,E1 -12574.02,E2 -12574.02} C_VEL
LIN {X 0,Y 368.924,Z 304.528,A -85,B 0,C 180,E1 -12577.605,E2 -12577.605} C_VEL
LIN {X 0,Y 368.966,Z 304.517,A -85,B 0,C 180,E1 -12581.107,E2 -12581.107} C_VEL
LIN {X 0,Y 368.997,Z 304.512,A -85,B 0,C 180,E1 -12584.535,E2 -12584.535} C_VEL
LIN {X 0,Y 369.004,Z 304.517,A -85,B 0,C 180,E1 -12587.907,E2 -12587.907} C_VEL
LIN {X 0,Y 369.228,Z 304.493,A -85,B 0,C 180,E1 -12591.802,E2 -12591.802} C_VEL
LIN {X 0,Y 369.143,Z 304.499,A -85,B 0,C 180,E1 -12594.538,E2 -12594.538} C_VEL
LIN {X 0,Y 369.316,Z 304.475,A -85,B 0,C 180,E1 -12597.819,E2 -12597.819} C_VEL
LIN {X 0,Y 369.456,Z 304.464,A -85,B 0,C 180,E1 -12600,E2 -12600} C_VEL
LIN {X 0,Y 369.316,Z 304.474,A -85,B 0,C 180,E1 -12602.181,E2 -12602.181} C_VEL
LIN {X 0,Y 369.206,Z 304.486,A -85,B 0,C 180,E1 -12606.558,E2 -12606.558} C_VEL
LIN {X 0,Y 369.138,Z 304.501,A -85,B 0,C 180,E1 -12608.761,E2 -12608.761} C_VEL
LIN {X 0,Y 369.005,Z 304.511,A -85,B 0,C 180,E1 -12612.094,E2 -12612.094} C_VEL
LIN {X 0,Y 368.998,Z 304.513,A -85,B 0,C 180,E1 -12615.465,E2 -12615.465} C_VEL
LIN {X 0,Y 368.983,Z 304.52,A -85,B 0,C 180,E1 -12618.893,E2 -12618.893} C_VEL
LIN {X 0,Y 368.925,Z 304.529,A -85,B 0,C 180,E1 -12622.396,E2 -12622.396} C_VEL
LIN {X 0,Y 369.001,Z 304.517,A -85,B 0,C 180,E1 -12625.98,E2 -12625.98} C_VEL
LIN {X 0,Y 368.96,Z 304.521,A -85,B 0,C 180,E1 -12628.811,E2 -12628.811} C_VEL
LIN {X 0,Y 368.899,Z 304.527,A -85,B 0,C 180,E1 -12632.238,E2 -12632.238} C_VEL
LIN {X 0,Y 368.93,Z 304.529,A -85,B 0,C 180,E1 -12635.002,E2 -12635.002} C_VEL
LIN {X 0,Y 368.909,Z 304.529,A -85,B 0,C 180,E1 -12638.64,E2 -12638.64} C_VEL
LIN {X 0,Y 368.883,Z 304.531,A -85,B 0,C 180,E1 -12642.01,E2 -12642.01} C_VEL
LIN {X 0,Y 368.881,Z 304.534,A -85,B 0,C 180,E1 -12645.176,E2 -12645.176} C_VEL
LIN {X 0,Y 368.884,Z 304.534,A -85,B 0,C 180,E1 -12648.178,E2 -12648.178} C_VEL
LIN {X 0,Y 368.909,Z 304.534,A -85,B 0,C 180,E1 -12651.36,E2 -12651.36} C_VEL
LIN {X 0,Y 368.939,Z 304.526,A -85,B 0,C 180,E1 -12655.147,E2 -12655.147} C_VEL
LIN {X 0,Y 368.932,Z 304.64,A -85,B 0,C 180,E1 -12659.047,E2 -12659.047} C_VEL
LIN {X 0,Y 371.62,Z 315.941,A -85,B 0,C 180,E1 -12662.026,E2 -12662.026} C_VEL
LIN {X 0,Y 373.452,Z 325.236,A -85,B 0,C 180,E1 -12664.352,E2 -12664.352} C_VEL
LIN {X 0,Y 373.22,Z 329.326,A -85,B 0,C 180,E1 -12665.28,E2 -12665.28} C_VEL
LIN {X 0,Y 372.229,Z 339.399,A -85,B 0,C 180,E1 -12667.512,E2 -12667.512} C_VEL
LIN {X 0,Y 376.902,Z 363.345,A -85,B 0,C 180,E1 -12668.35,E2 -12668.35} C_VEL
LIN {X 0,Y 378.544,Z 375.051,A -85,B 0,C 180,E1 -12668.704,E2 -12668.704} C_VEL
LIN {X 0,Y 377.162,Z 448.907,A -85,B 0,C 180,E1 -12670.154,E2 -12670.154} C_VEL
LIN {X 0,Y 376.342,Z 462.578,A -85,B 0,C 180,E1 -12670.642,E2 -12670.642} C_VEL
LIN {X 0,Y 375.441,Z 474.877,A -85,B 0,C 180,E1 -12671.302,E2 -12671.302} C_VEL
LIN {X 0,Y 374.155,Z 487.483,A -85,B 0,C 180,E1 -12672.228,E2 -12672.228} C_VEL
LIN {X 0,Y 372.966,Z 498.707,A -85,B 0,C 180,E1 -12673.3,E2 -12673.3} C_VEL
LIN {X 0,Y 371.75,Z 508.85,A -85,B 0,C 180,E1 -12674.512,E2 -12674.512} C_VEL
LIN {X 0,Y 370.824,Z 517.18,A -85,B 0,C 180,E1 -12675.736,E2 -12675.736} C_VEL
LIN {X 0,Y 369.702,Z 526.246,A -85,B 0,C 180,E1 -12677.372,E2 -12677.372} C_VEL
LIN {X 0,Y 368.749,Z 533.573,A -85,B 0,C 180,E1 -12679.012,E2 -12679.012} C_VEL
LIN {X 0,Y 368.143,Z 539.469,A -85,B 0,C 180,E1 -12680.661,E2 -12680.661} C_VEL
LIN {X 0,Y 367.73,Z 544.136,A -85,B 0,C 180,E1 -12682.311,E2 -12682.311} C_VEL
LIN {X 0,Y 367.507,Z 547.679,A -85,B 0,C 180,E1 -12683.946,E2 -12683.946} C_VEL
LIN {X 0,Y 367.457,Z 550.288,A -85,B 0,C 180,E1 -12685.612,E2 -12685.612} C_VEL
LIN {X 0,Y 367.382,Z 551.506,A -85,B 0,C 180,E1 -12686.71,E2 -12686.71} C_VEL
LIN {X 0,Y 367.396,Z 552.288,A -85,B 0,C 180,E1 -12687.807,E2 -12687.807} C_VEL
LIN {X 0,Y 367.457,Z 552.673,A -85,B 0,C 180,E1 -12688.904,E2 -12688.904} C_VEL
LIN {X 0,Y 367.505,Z 552.672,A -85,B 0,C 180,E1 -12690,E2 -12690} C_VEL
LIN {X 0,Y 367.488,Z 552.282,A -85,B 0,C 180,E1 -12691.095,E2 -12691.095} C_VEL
LIN {X 0,Y 367.425,Z 551.46,A -85,B 0,C 180,E1 -12692.192,E2 -12692.192} C_VEL
LIN {X 0,Y 367.494,Z 548.575,A -85,B 0,C 180,E1 -12694.387,E2 -12694.387} C_VEL
LIN {X 0,Y 367.514,Z 545.187,A -85,B 0,C 180,E1 -12696.064,E2 -12696.064} C_VEL
LIN {X 0,Y 367.693,Z 540.839,A -85,B 0,C 180,E1 -12697.689,E2 -12697.689} C_VEL
LIN {X 0,Y 368.016,Z 535.217,A -85,B 0,C 180,E1 -12699.341,E2 -12699.341} C_VEL
LIN {X 0,Y 368.515,Z 528.183,A -85,B 0,C 180,E1 -12700.994,E2 -12700.994} C_VEL
LIN {X 0,Y 369.36,Z 519.365,A -85,B 0,C 180,E1 -12702.639,E2 -12702.639} C_VEL
LIN {X 0,Y 370.255,Z 509.332,A -85,B 0,C 180,E1 -12704.145,E2 -12704.145} C_VEL
LIN {X 0,Y 371.004,Z 499.079,A -85,B 0,C 180,E1 -12705.379,E2 -12705.379} C_VEL
LIN {X 0,Y 371.929,Z 487.696,A -85,B 0,C 180,E1 -12706.465,E2 -12706.465} C_VEL
LIN {X 0,Y 372.866,Z 475.897,A -85,B 0,C 180,E1 -12707.34,E2 -12707.34} C_VEL
LIN {X 0,Y 373.583,Z 463.734,A -85,B 0,C 180,E1 -12708.012,E2 -12708.012} C_VEL
LIN {X 0,Y 374.217,Z 450.281,A -85,B 0,C 180,E1 -12708.512,E2 -12708.512} C_VEL
LIN {X 0,Y 374.602,Z 427.424,A -85,B 0,C 180,E1 -12708.99,E2 -12708.99} C_VEL
LIN {X 0,Y 375.247,Z 372.158,A -85,B 0,C 180,E1 -12710.046,E2 -12710.046} C_VEL
LIN {X 0,Y 370.723,Z 339.825,A -85,B 0,C 180,E1 -12710.92,E2 -12710.92} C_VEL
LIN {X 0,Y 372.012,Z 324.345,A -85,B 0,C 180,E1 -12714.261,E2 -12714.261} C_VEL
LIN {X 0,Y 372.172,Z 321.043,A -85,B 0,C 180,E1 -12714.984,E2 -12714.984} C_VEL
LIN {X 0,Y 370.025,Z 309.363,A -85,B 0,C 180,E1 -12717.731,E2 -12717.731} C_VEL
LIN {X 0,Y 368.985,Z 304.524,A -85,B 0,C 180,E1 -12718.959,E2 -12718.959} C_VEL
LIN {X 0,Y 368.898,Z 304.535,A -85,B 0,C 180,E1 -12722.237,E2 -12722.237} C_VEL
LIN {X 0,Y 368.928,Z 304.526,A -85,B 0,C 180,E1 -12725.001,E2 -12725.001} C_VEL
LIN {X 0,Y 368.905,Z 304.532,A -85,B 0,C 180,E1 -12728.639,E2 -12728.639} C_VEL
LIN {X 0,Y 368.88,Z 304.534,A -85,B 0,C 180,E1 -12732.009,E2 -12732.009} C_VEL
LIN {X 0,Y 368.878,Z 304.533,A -85,B 0,C 180,E1 -12735.175,E2 -12735.175} C_VEL
LIN {X 0,Y 368.881,Z 304.534,A -85,B 0,C 180,E1 -12738.177,E2 -12738.177} C_VEL
LIN {X 0,Y 368.906,Z 304.529,A -85,B 0,C 180,E1 -12741.359,E2 -12741.359} C_VEL
LIN {X 0,Y 368.933,Z 304.528,A -85,B 0,C 180,E1 -12745.146,E2 -12745.146} C_VEL
LIN {X 0,Y 368.926,Z 304.531,A -85,B 0,C 180,E1 -12749.046,E2 -12749.046} C_VEL
LIN {X 0,Y 368.959,Z 304.526,A -85,B 0,C 180,E1 -12752.796,E2 -12752.796} C_VEL
LIN {X 0,Y 368.941,Z 304.524,A -85,B 0,C 180,E1 -12756.112,E2 -12756.112} C_VEL
LIN {X 0,Y 368.932,Z 304.525,A -85,B 0,C 180,E1 -12759.947,E2 -12759.947} C_VEL
LIN {X 0,Y 368.972,Z 304.526,A -85,B 0,C 180,E1 -12763.398,E2 -12763.398} C_VEL
LIN {X 0,Y 369.053,Z 304.511,A -85,B 0,C 180,E1 -12766.79,E2 -12766.79} C_VEL
LIN {X 0,Y 369.063,Z 304.509,A -85,B 0,C 180,E1 -12770.131,E2 -12770.131} C_VEL
LIN {X 0,Y 369.158,Z 304.497,A -85,B 0,C 180,E1 -12772.341,E2 -12772.341} C_VEL
LIN {X 0,Y 369.137,Z 304.499,A -85,B 0,C 180,E1 -12774.537,E2 -12774.537} C_VEL
LIN {X 0,Y 369.311,Z 304.483,A -85,B 0,C 180,E1 -12777.819,E2 -12777.819} C_VEL
LIN {X 0,Y 369.451,Z 304.464,A -85,B 0,C 180,E1 -12780,E2 -12780} C_VEL
LIN {X 0,Y 369.312,Z 304.48,A -85,B 0,C 180,E1 -12782.181,E2 -12782.181} C_VEL
LIN {X 0,Y 369.173,Z 304.496,A -85,B 0,C 180,E1 -12786.559,E2 -12786.559} C_VEL
LIN {X 0,Y 369.062,Z 304.514,A -85,B 0,C 180,E1 -12789.868,E2 -12789.868} C_VEL
LIN {X 0,Y 369.032,Z 304.516,A -85,B 0,C 180,E1 -12793.772,E2 -12793.772} C_VEL
LIN {X 0,Y 368.996,Z 304.519,A -85,B 0,C 180,E1 -12797.768,E2 -12797.768} C_VEL
LIN {X 0,Y 368.904,Z 304.528,A -85,B 0,C 180,E1 -12801.221,E2 -12801.221} C_VEL
LIN {X 0,Y 368.948,Z 304.526,A -85,B 0,C 180,E1 -12804.776,E2 -12804.776} C_VEL
LIN {X 0,Y 368.963,Z 304.522,A -85,B 0,C 180,E1 -12807.203,E2 -12807.203} C_VEL
LIN {X 0,Y 368.914,Z 304.527,A -85,B 0,C 180,E1 -12809.69,E2 -12809.69} C_VEL
LIN {X 0,Y 368.892,Z 304.532,A -85,B 0,C 180,E1 -12813.043,E2 -12813.043} C_VEL
LIN {X 0,Y 368.912,Z 304.529,A -85,B 0,C 180,E1 -12816.197,E2 -12816.197} C_VEL
LIN {X 0,Y 368.897,Z 304.534,A -85,B 0,C 180,E1 -12818.954,E2 -12818.954} C_VEL
LIN {X 0,Y 368.876,Z 304.532,A -85,B 0,C 180,E1 -12822.01,E2 -12822.01} C_VEL
LIN {X 0,Y 368.875,Z 304.537,A -85,B 0,C 180,E1 -12825.176,E2 -12825.176} C_VEL
LIN {X 0,Y 368.865,Z 304.533,A -85,B 0,C 180,E1 -12828.176,E2 -12828.176} C_VEL
LIN {X 0,Y 368.874,Z 304.536,A -85,B 0,C 180,E1 -12831.366,E2 -12831.366} C_VEL
LIN {X 0,Y 368.933,Z 304.531,A -85,B 0,C 180,E1 -12835.147,E2 -12835.147} C_VEL
LIN {X 0,Y 368.909,Z 304.531,A -85,B 0,C 180,E1 -12839.045,E2 -12839.045} C_VEL
LIN {X 0,Y 368.904,Z 304.534,A -85,B 0,C 180,E1 -12841.558,E2 -12841.558} C_VEL
LIN {X 0,Y 368.895,Z 304.533,A -85,B 0,C 180,E1 -12845.221,E2 -12845.221} C_VEL
LIN {X 0,Y 368.918,Z 304.534,A -85,B 0,C 180,E1 -12847.605,E2 -12847.605} C_VEL
LIN {X 0,Y 368.953,Z 304.524,A -85,B 0,C 180,E1 -12851.106,E2 -12851.106} C_VEL
LIN {X 0,Y 368.996,Z 304.521,A -85,B 0,C 180,E1 -12854.536,E2 -12854.536} C_VEL
LIN {X 0,Y 369.093,Z 304.551,A -85,B 0,C 180,E1 -12856.697,E2 -12856.697} C_VEL
LIN {X 0,Y 370.832,Z 314.205,A -85,B 0,C 180,E1 -12859.162,E2 -12859.162} C_VEL
LIN {X 0,Y 372.903,Z 322.492,A -85,B 0,C 180,E1 -12859.447,E2 -12859.447} C_VEL
LIN {X 0,Y 375.782,Z 338.872,A -85,B 0,C 180,E1 -12859.911,E2 -12859.911} C_VEL
LIN {X 0,Y 374.481,Z 421.542,A -85,B 0,C 180,E1 -12861.501,E2 -12861.501} C_VEL
LIN {X 0,Y 374.038,Z 434.727,A -85,B 0,C 180,E1 -12861.967,E2 -12861.967} C_VEL
